C05464=1030.922,10.117,408.960,168.211,43.114,158.030
C05465=1030.915,9.868,408.976,168.209,43.115,158.030
C05466=1030.909,9.618,408.991,168.206,43.117,158.030
C05467=1030.902,9.369,409.006,168.203,43.118,158.030
C05468=1030.896,9.120,409.020,168.200,43.120,158.030
C05469=1030.890,8.870,409.035,168.199,43.121,158.030
C05470=1030.884,8.620,409.050,168.196,43.122,158.030
C05471=1030.877,8.371,409.066,168.193,43.124,158.030
C05472=1030.871,8.122,409.081,168.191,43.125,158.031
C05473=1030.864,7.872,409.096,168.189,43.126,158.031
C05474=1030.858,7.623,409.110,168.186,43.128,158.031
C05475=1030.852,7.374,409.125,168.184,43.129,158.031
C05476=1030.846,7.124,409.140,168.181,43.131,158.031
C05477=1030.839,6.874,409.155,168.179,43.132,158.031
C05478=1030.833,6.625,409.170,168.177,43.134,158.031
C05479=1030.826,6.375,409.185,168.174,43.135,158.031
C05480=1030.821,6.126,409.199,168.171,43.136,158.031
C05481=1030.814,5.876,409.214,168.169,43.138,158.031
C05482=1030.808,5.627,409.229,168.167,43.139,158.031
C05483=1030.801,5.377,409.244,168.164,43.141,158.031
C05484=1030.795,5.128,409.260,168.161,43.142,158.031
C05485=1030.789,4.879,409.275,168.159,43.143,158.031
C05486=1030.783,4.629,409.290,168.157,43.145,158.031
C05487=1030.776,4.380,409.304,168.154,43.146,158.031
C05488=1030.770,4.130,409.319,168.152,43.148,158.032
C05489=1030.764,3.881,409.334,168.150,43.149,158.032
C05490=1030.758,3.631,409.349,168.147,43.150,158.032
C05491=1030.751,3.382,409.364,168.145,43.152,158.032
C05492=1030.745,3.132,409.379,168.142,43.153,158.032
C05493=1030.739,2.883,409.393,168.139,43.154,158.032
C05494=1030.733,2.633,409.408,168.138,43.156,158.032
C05495=1030.727,2.383,409.423,168.135,43.157,158.032
C05496=1030.721,2.134,409.437,168.132,43.159,158.032
C05497=1030.715,1.885,409.452,168.129,43.160,158.032
C05498=1030.708,1.635,409.467,168.128,43.161,158.032
C05499=1030.702,1.385,409.482,168.125,43.163,158.032
C05500=1030.696,1.136,409.497,168.122,43.164,158.032
C05501=1030.690,0.887,409.512,168.120,43.165,158.032
C05502=1030.683,0.637,409.526,168.118,43.167,158.032
C05503=1030.677,0.388,409.541,168.115,43.168,158.032
C05504=1030.671,0.138,409.556,168.113,43.169,158.033
C05505=1030.665,-0.111,409.571,168.110,43.171,158.033
C05506=1030.659,-0.361,409.585,168.107,43.172,158.033
C05507=1030.653,-0.611,409.600,168.106,43.173,158.033
C05508=1030.646,-0.860,409.615,168.103,43.175,158.033
C05509=1030.641,-1.109,409.629,168.100,43.176,158.033
C05510=1030.634,-1.359,409.644,168.097,43.177,158.033
C05511=1030.628,-1.608,409.659,168.096,43.179,158.033
C05512=1030.622,-1.857,409.674,168.093,43.180,158.033
C05513=1030.616,-2.108,409.688,168.090,43.181,158.033
C05514=1030.609,-2.357,409.702,168.088,43.183,158.033
C05515=1030.603,-2.606,409.717,168.085,43.184,158.033
C05516=1030.597,-2.856,409.732,168.083,43.185,158.033
C05517=1030.591,-3.105,409.746,168.081,43.187,158.033
C05518=1030.585,-3.355,409.761,168.078,43.188,158.033
C05519=1030.578,-3.605,409.776,168.075,43.189,158.033
C05520=1030.572,-3.887,409.792,168.073,43.191,158.033
C05521=1030.565,-4.170,409.809,168.070,43.193,158.034
C05522=1030.558,-4.454,409.825,168.067,43.194,158.034
C05523=1030.550,-4.736,409.840,168.064,43.196,158.034
C05524=1030.544,-4.986,409.855,168.062,43.197,158.034
C05525=1030.538,-5.235,409.870,168.059,43.199,158.034
C05526=1030.531,-5.485,409.884,168.056,43.200,158.034
C05527=1030.525,-5.734,409.899,168.054,43.202,158.034
C05528=1030.518,-5.984,409.912,168.052,43.204,158.034
C05529=1030.512,-6.233,409.927,168.049,43.205,158.034
C05530=1030.506,-6.483,409.942,168.046,43.207,158.034
C05531=1030.500,-6.732,409.955,168.043,43.208,158.034
C05532=1030.493,-6.982,409.970,168.042,43.210,158.034
C05533=1030.487,-7.232,409.984,168.039,43.211,158.034
C05534=1030.481,-7.481,409.998,168.036,43.213,158.035
C05535=1030.475,-7.731,410.012,168.034,43.214,158.035
C05536=1030.468,-7.980,410.026,168.032,43.215,158.035
C05537=1030.462,-8.229,410.041,168.029,43.217,158.035
C05538=1030.456,-8.479,410.055,168.026,43.218,158.035
C05539=1030.449,-8.728,410.069,168.024,43.220,158.035
C05540=1030.443,-8.978,410.084,168.021,43.221,158.035
C05541=1030.437,-9.227,410.098,168.019,43.223,158.035
C05542=1030.431,-9.477,410.112,168.016,43.224,158.035
C05543=1030.424,-9.726,410.126,168.014,43.226,158.035
C05544=1030.418,-9.976,410.140,168.011,43.227,158.035
C05545=1030.412,-10.225,410.155,168.009,43.229,158.035
C05546=1030.405,-10.475,410.168,168.006,43.230,158.035
C05547=1030.400,-10.724,410.183,168.004,43.232,158.035
C05548=1030.393,-10.974,410.197,168.001,43.233,158.035
C05549=1030.387,-11.224,410.210,167.998,43.235,158.036
C05550=1030.381,-11.473,410.225,167.996,43.236,158.036
C05551=1030.375,-11.723,410.239,167.993,43.237,158.036
C05552=1030.368,-11.972,410.254,167.991,43.239,158.036
C05553=1030.362,-12.222,410.267,167.988,43.240,158.036
C05554=1030.356,-12.471,410.282,167.985,43.242,158.036
C05555=1030.349,-12.720,410.295,167.983,43.243,158.036
C05556=1030.343,-12.971,410.309,167.981,43.245,158.036
C05557=1030.338,-13.220,410.324,167.978,43.246,158.036
C05558=1030.331,-13.470,410.338,167.975,43.248,158.036
C05559=1030.325,-13.719,410.352,167.973,43.249,158.036
C05560=1030.318,-13.969,410.366,167.971,43.250,158.036
C05561=1030.313,-14.218,410.380,167.968,43.252,158.036
C05562=1030.306,-14.467,410.394,167.965,43.253,158.036
C05563=1030.300,-14.717,410.408,167.963,43.255,158.036
C05564=1030.295,-14.967,410.422,167.961,43.256,158.036
C05565=1030.288,-15.216,410.436,167.958,43.258,158.037
C05566=1030.282,-15.466,410.450,167.955,43.259,158.037
C05567=1030.275,-15.716,410.464,167.952,43.260,158.037
C05568=1030.269,-15.965,410.477,167.950,43.262,158.037
C05569=1030.263,-16.215,410.491,167.947,43.264,158.037
C05570=1030.256,-16.464,410.505,167.945,43.265,158.037
C05571=1030.250,-16.713,410.518,167.943,43.266,158.037
C05572=1030.244,-16.963,410.533,167.940,43.268,158.037
C05573=1030.238,-17.213,410.546,167.937,43.269,158.037
C05574=1030.231,-17.463,410.559,167.934,43.271,158.037
C05575=1030.225,-17.711,410.574,167.932,43.273,158.037
C05576=1030.219,-17.961,410.588,167.930,43.274,158.037
C05577=1030.212,-18.211,410.601,167.927,43.275,158.037
C05578=1030.207,-18.460,410.615,167.924,43.277,158.038
C05579=1030.200,-18.710,410.628,167.922,43.278,158.038
C05580=1030.194,-18.960,410.642,167.919,43.280,158.038
C05581=1030.187,-19.209,410.657,167.916,43.281,158.038
C05582=1030.181,-19.458,410.670,167.913,43.283,158.038
C05583=1030.175,-19.708,410.683,167.912,43.285,158.038
C05584=1030.168,-19.989,410.698,167.908,43.286,158.038
C05585=1030.161,-20.271,410.714,167.905,43.288,158.038
C05586=1030.153,-20.552,410.729,167.903,43.290,158.038
C05587=1030.147,-20.834,410.744,167.900,43.291,158.038
C05588=1030.141,-21.083,410.758,167.897,43.293,158.038
C05589=1030.134,-21.333,410.772,167.895,43.295,158.038
C05590=1030.128,-21.583,410.785,167.892,43.296,158.038
C05591=1030.122,-21.832,410.799,167.889,43.298,158.038
C05592=1030.115,-22.082,410.813,167.886,43.299,158.038
C05593=1030.109,-22.331,410.827,167.885,43.301,158.039
C05594=1030.103,-22.580,410.840,167.882,43.302,158.039
C05595=1030.098,-22.830,410.854,167.879,43.304,158.039
C05596=1030.091,-23.080,410.867,167.876,43.305,158.039
C05597=1030.085,-23.329,410.881,167.874,43.307,158.039
C05598=1030.078,-23.578,410.894,167.871,43.308,158.039
C05599=1030.072,-23.828,410.908,167.868,43.310,158.039
C05600=1030.066,-24.078,410.922,167.866,43.311,158.039
C05601=1030.060,-24.327,410.935,167.864,43.313,158.039
C05602=1030.055,-24.577,410.948,167.861,43.314,158.039
C05603=1030.048,-24.827,410.962,167.858,43.316,158.039
C05604=1030.042,-25.076,410.975,167.855,43.317,158.039
C05605=1030.035,-25.326,410.988,167.853,43.319,158.039
C05606=1030.030,-25.575,411.002,167.850,43.320,158.039
C05607=1030.023,-25.825,411.016,167.848,43.322,158.040
C05608=1030.017,-26.074,411.029,167.845,43.323,158.040
C05609=1030.011,-26.324,411.042,167.843,43.325,158.040
C05610=1030.005,-26.573,411.056,167.840,43.326,158.040
C05611=1029.998,-26.823,411.070,167.837,43.328,158.040
C05612=1029.992,-27.072,411.083,167.834,43.329,158.040
C05613=1029.986,-27.322,411.095,167.832,43.331,158.040
C05614=1029.980,-27.572,411.109,167.829,43.332,158.040
C05615=1029.973,-27.822,411.122,167.826,43.334,158.040
C05616=1029.967,-28.071,411.136,167.825,43.336,158.040
C05617=1029.961,-28.320,411.149,167.822,43.337,158.040
C05618=1029.955,-28.570,411.161,167.819,43.339,158.040
C05619=1029.948,-28.820,411.175,167.816,43.341,158.040
C05620=1029.942,-29.069,411.188,167.814,43.342,158.040
C05621=1029.936,-29.318,411.202,167.811,43.344,158.041
C05622=1029.930,-29.568,411.214,167.808,43.345,158.041
C05623=1029.924,-29.818,411.227,167.805,43.347,158.041
C05624=1029.917,-30.068,411.241,167.803,43.349,158.041
C05625=1029.910,-30.317,411.254,167.800,43.350,158.041
C05626=1029.905,-30.567,411.267,167.797,43.352,158.041
C05627=1029.898,-30.816,411.280,167.795,43.354,158.041
C05628=1029.892,-31.065,411.293,167.792,43.355,158.041
C05629=1029.886,-31.315,411.306,167.789,43.357,158.041
C05630=1029.879,-31.565,411.320,167.787,43.358,158.041
C05631=1029.873,-31.814,411.333,167.785,43.359,158.041
C05632=1029.867,-32.064,411.346,167.782,43.361,158.041
C05633=1029.861,-32.314,411.359,167.779,43.363,158.041
C05634=1029.855,-32.563,411.372,167.777,43.364,158.042
C05635=1029.849,-32.813,411.385,167.774,43.366,158.042
C05636=1029.842,-33.063,411.398,167.771,43.367,158.042
C05637=1029.836,-33.313,411.411,167.768,43.369,158.042
C05638=1029.830,-33.562,411.424,167.766,43.370,158.042
C05639=1029.824,-33.811,411.437,167.763,43.372,158.042
C05640=1029.818,-34.061,411.450,167.760,43.374,158.042
C05641=1029.812,-34.310,411.463,167.757,43.375,158.042
C05642=1029.806,-34.560,411.476,167.755,43.377,158.042
C05643=1029.800,-34.809,411.489,167.752,43.378,158.042
C05644=1029.794,-35.059,411.502,167.749,43.380,158.042
C05645=1029.787,-35.308,411.515,167.747,43.382,158.042
C05646=1029.781,-35.558,411.528,167.745,43.383,158.042
C05647=1029.775,-35.808,411.541,167.742,43.385,158.042
C05648=1029.768,-36.088,411.556,167.738,43.386,158.042
C05649=1029.761,-36.369,411.570,167.736,43.388,158.043
C05650=1029.754,-36.650,411.584,167.733,43.390,158.043
C05651=1029.747,-36.930,411.599,167.729,43.392,158.043
C05652=1029.741,-37.180,411.611,167.727,43.393,158.043
C05653=1029.735,-37.429,411.624,167.724,43.395,158.043
C05654=1029.729,-37.679,411.637,167.722,43.397,158.043
C05655=1029.723,-37.928,411.650,167.719,43.398,158.043
C05656=1029.717,-38.178,411.663,167.717,43.400,158.043
C05657=1029.711,-38.427,411.676,167.714,43.401,158.043
C05658=1029.705,-38.677,411.689,167.711,43.403,158.043
C05659=1029.699,-38.927,411.702,167.708,43.404,158.043
C05660=1029.693,-39.176,411.715,167.706,43.406,158.043
C05661=1029.686,-39.426,411.726,167.703,43.408,158.043
C05662=1029.680,-39.675,411.740,167.700,43.410,158.044
C05663=1029.674,-39.925,411.752,167.698,43.411,158.044
C05664=1029.668,-40.175,411.765,167.695,43.413,158.044
C05665=1029.661,-40.424,411.778,167.692,43.415,158.044
C05666=1029.655,-40.674,411.790,167.689,43.416,158.044
C05667=1029.649,-40.924,411.803,167.687,43.418,158.044
C05668=1029.642,-41.173,411.815,167.684,43.420,158.044
C05669=1029.636,-41.423,411.828,167.682,43.422,158.044
C05670=1029.630,-41.672,411.840,167.679,43.423,158.044
C05671=1029.624,-41.922,411.852,167.676,43.425,158.044
C05672=1029.618,-42.171,411.866,167.673,43.427,158.044
C05673=1029.612,-42.421,411.878,167.671,43.428,158.044
C05674=1029.606,-42.671,411.891,167.668,43.430,158.045
C05675=1029.599,-42.921,411.903,167.665,43.432,158.045
C05676=1029.593,-43.170,411.916,167.663,43.433,158.045
C05677=1029.587,-43.420,411.929,167.660,43.435,158.045
C05678=1029.580,-43.669,411.940,167.657,43.436,158.045
C05679=1029.574,-43.919,411.953,167.655,43.438,158.045
C05680=1029.569,-44.169,411.966,167.652,43.440,158.045
C05681=1029.562,-44.418,411.978,167.649,43.441,158.045
C05682=1029.556,-44.668,411.991,167.646,43.443,158.045
C05683=1029.550,-44.918,412.003,167.644,43.444,158.045
C05684=1029.543,-45.167,412.015,167.641,43.446,158.045
C05685=1029.538,-45.417,412.028,167.638,43.448,158.045
C05686=1029.532,-45.666,412.040,167.635,43.449,158.045
C05687=1029.525,-45.915,412.053,167.633,43.451,158.046
C05688=1029.519,-46.165,412.065,167.630,43.453,158.046
C05689=1029.513,-46.415,412.078,167.626,43.455,158.046
C05690=1029.507,-46.665,412.090,167.624,43.456,158.046
C05691=1029.501,-46.915,412.102,167.621,43.458,158.046
C05692=1029.495,-47.165,412.115,167.618,43.460,158.046
C05693=1029.489,-47.413,412.127,167.615,43.461,158.046
C05694=1029.483,-47.663,412.139,167.613,43.463,158.046
C05695=1029.477,-47.913,412.152,167.610,43.465,158.046
C05696=1029.470,-48.163,412.164,167.607,43.466,158.046
C05697=1029.464,-48.413,412.176,167.605,43.468,158.046
C05698=1029.458,-48.662,412.189,167.602,43.470,158.046
C05699=1029.452,-48.911,412.201,167.599,43.471,158.046
C05700=1029.446,-49.161,412.214,167.597,43.473,158.046
C05701=1029.439,-49.410,412.226,167.594,43.475,158.047
C05702=1029.434,-49.660,412.238,167.591,43.476,158.047
C05703=1029.428,-49.910,412.251,167.588,43.478,158.047
C05704=1029.422,-50.159,412.262,167.586,43.480,158.047
C05705=1029.416,-50.409,412.275,167.583,43.481,158.047
C05706=1029.410,-50.659,412.287,167.580,43.483,158.047
C05707=1029.403,-50.909,412.299,167.578,43.485,158.047
C05708=1029.397,-51.158,412.311,167.575,43.487,158.047
C05709=1029.391,-51.408,412.323,167.572,43.489,158.047
C05710=1029.384,-51.658,412.335,167.570,43.491,158.047
C05711=1029.378,-51.907,412.347,167.567,43.492,158.047
C05712=1029.372,-52.188,412.360,167.563,43.494,158.048
C05713=1029.364,-52.469,412.374,167.561,43.496,158.048
C05714=1029.357,-52.750,412.387,167.557,43.498,158.048
C05715=1029.350,-53.031,412.401,167.554,43.500,158.048
C05716=1029.343,-53.281,412.412,167.551,43.502,158.048
C05717=1029.338,-53.530,412.424,167.548,43.504,158.048
C05718=1029.331,-53.780,412.436,167.546,43.506,158.048
C05719=1029.325,-54.029,412.448,167.543,43.508,158.048
C05720=1029.318,-54.280,412.459,167.540,43.510,158.048
C05721=1029.313,-54.529,412.471,167.537,43.511,158.048
C05722=1029.306,-54.778,412.483,167.535,43.513,158.049
C05723=1029.300,-55.028,412.495,167.532,43.515,158.049
C05724=1029.293,-55.278,412.507,167.528,43.517,158.049
C05725=1029.288,-55.527,412.519,167.526,43.519,158.049
C05726=1029.282,-55.777,412.531,167.523,43.521,158.049
C05727=1029.275,-56.027,412.542,167.521,43.523,158.049
C05728=1029.269,-56.277,412.554,167.518,43.524,158.049
C05729=1029.263,-56.526,412.566,167.515,43.526,158.049
C05730=1029.257,-56.775,412.578,167.512,43.527,158.049
C05731=1029.250,-57.026,412.589,167.510,43.529,158.049
C05732=1029.244,-57.274,412.601,167.506,43.531,158.049
C05733=1029.238,-57.524,412.613,167.503,43.533,158.050
C05734=1029.232,-57.774,412.625,167.501,43.535,158.050
C05735=1029.226,-58.023,412.636,167.498,43.537,158.050
C05736=1029.220,-58.274,412.648,167.496,43.539,158.050
C05737=1029.214,-58.523,412.660,167.493,43.541,158.050
C05738=1029.208,-58.772,412.672,167.490,43.542,158.050
C05739=1029.201,-59.022,412.683,167.487,43.544,158.050
C05740=1029.195,-59.272,412.695,167.484,43.546,158.050
C05741=1029.190,-59.522,412.706,167.481,43.548,158.050
C05742=1029.183,-59.771,412.718,167.478,43.550,158.050
C05743=1029.176,-60.021,412.730,167.476,43.552,158.051
C05744=1029.171,-60.270,412.741,167.473,43.554,158.051
C05745=1029.164,-60.520,412.753,167.470,43.555,158.051
C05746=1029.159,-60.770,412.765,167.468,43.557,158.051
C05747=1029.152,-61.019,412.777,167.465,43.559,158.051
C05748=1029.146,-61.270,412.788,167.461,43.561,158.051
C05749=1029.140,-61.519,412.799,167.459,43.562,158.051
C05750=1029.134,-61.769,412.811,167.456,43.564,158.051
C05751=1029.128,-62.018,412.823,167.453,43.566,158.051
C05752=1029.122,-62.268,412.834,167.451,43.567,158.051
C05753=1029.115,-62.518,412.846,167.448,43.569,158.051
C05754=1029.110,-62.767,412.857,167.445,43.571,158.051
C05755=1029.104,-63.017,412.869,167.442,43.573,158.052
C05756=1029.098,-63.267,412.880,167.439,43.575,158.052
C05757=1029.091,-63.516,412.892,167.436,43.577,158.052
C05758=1029.086,-63.766,412.903,167.434,43.579,158.052
C05759=1029.079,-64.015,412.915,167.431,43.580,158.052
C05760=1029.074,-64.265,412.927,167.428,43.582,158.052
C05761=1029.068,-64.515,412.938,167.426,43.584,158.052
C05762=1029.061,-64.764,412.949,167.423,43.586,158.052
C05763=1029.055,-65.014,412.961,167.419,43.588,158.052
C05764=1029.049,-65.263,412.972,167.417,43.590,158.052
C05765=1029.043,-65.514,412.984,167.414,43.591,158.052
C05766=1029.038,-65.763,412.995,167.411,43.593,158.052
C05767=1029.031,-66.013,413.007,167.409,43.595,158.053
C05768=1029.025,-66.262,413.018,167.406,43.597,158.053
C05769=1029.019,-66.512,413.029,167.403,43.599,158.053
C05770=1029.014,-66.761,413.041,167.400,43.601,158.053
C05771=1029.007,-67.012,413.052,167.397,43.602,158.053
C05772=1029.002,-67.261,413.063,167.394,43.604,158.053
C05773=1028.995,-67.511,413.075,167.391,43.606,158.053
C05774=1028.989,-67.760,413.086,167.389,43.607,158.053
C05775=1028.983,-68.010,413.097,167.386,43.609,158.053
C05776=1028.976,-68.292,413.111,167.383,43.611,158.053
C05777=1028.970,-68.574,413.124,167.380,43.613,158.053
C05778=1028.964,-68.856,413.136,167.376,43.615,158.054
C05779=1028.956,-69.139,413.149,167.374,43.617,158.054
C05780=1028.951,-69.389,413.160,167.370,43.619,158.054
C05781=1028.945,-69.639,413.172,167.367,43.621,158.054
C05782=1028.939,-69.888,413.183,167.364,43.622,158.054
C05783=1028.932,-70.138,413.194,167.362,43.624,158.054
C05784=1028.927,-70.387,413.205,167.359,43.626,158.054
C05785=1028.921,-70.637,413.216,167.357,43.628,158.054
C05786=1028.915,-70.887,413.229,167.354,43.630,158.054
C05787=1028.909,-71.136,413.240,167.350,43.631,158.054
C05788=1028.903,-71.386,413.251,167.347,43.633,158.054
C05789=1028.897,-71.636,413.262,167.345,43.635,158.054
C05790=1028.891,-71.885,413.273,167.342,43.637,158.055
C05791=1028.885,-72.136,413.284,167.339,43.639,158.055
C05792=1028.879,-72.384,413.295,167.337,43.640,158.055
C05793=1028.874,-72.634,413.307,167.334,43.642,158.055
C05794=1028.868,-72.884,413.318,167.330,43.644,158.055
C05795=1028.862,-73.134,413.329,167.328,43.646,158.055
C05796=1028.856,-73.383,413.340,167.325,43.648,158.055
C05797=1028.850,-73.633,413.351,167.322,43.649,158.055
C05798=1028.844,-73.883,413.362,167.320,43.651,158.055
C05799=1028.838,-74.132,413.374,167.317,43.653,158.055
C05800=1028.832,-74.381,413.384,167.314,43.655,158.055
C05801=1028.826,-74.632,413.396,167.311,43.657,158.055
C05802=1028.820,-74.881,413.407,167.308,43.659,158.055
C05803=1028.815,-75.131,413.417,167.305,43.661,158.056
C05804=1028.808,-75.381,413.428,167.303,43.663,158.056
C05805=1028.803,-75.631,413.439,167.300,43.664,158.056
C05806=1028.796,-75.880,413.449,167.296,43.667,158.056
C05807=1028.790,-76.130,413.460,167.294,43.668,158.056
C05808=1028.784,-76.380,413.471,167.291,43.670,158.056
C05809=1028.778,-76.629,413.482,167.288,43.672,158.056
C05810=1028.772,-76.879,413.493,167.285,43.674,158.056
C05811=1028.766,-77.129,413.504,167.282,43.676,158.056
C05812=1028.761,-77.378,413.515,167.280,43.678,158.056
C05813=1028.754,-77.628,413.525,167.277,43.680,158.057
C05814=1028.748,-77.878,413.537,167.274,43.682,158.057
C05815=1028.742,-78.127,413.548,167.271,43.684,158.057
C05816=1028.736,-78.377,413.558,167.268,43.686,158.057
C05817=1028.731,-78.627,413.569,167.265,43.688,158.057
C05818=1028.725,-78.877,413.580,167.263,43.690,158.057
C05819=1028.719,-79.127,413.591,167.260,43.692,158.057
C05820=1028.712,-79.376,413.601,167.256,43.693,158.057
C05821=1028.707,-79.625,413.612,167.253,43.695,158.057
C05822=1028.701,-79.876,413.622,167.251,43.697,158.057
C05823=1028.695,-80.126,413.633,167.248,43.699,158.057
C05824=1028.688,-80.375,413.644,167.245,43.701,158.058
C05825=1028.683,-80.624,413.654,167.242,43.703,158.058
C05826=1028.677,-80.874,413.665,167.239,43.705,158.058
C05827=1028.670,-81.124,413.675,167.237,43.707,158.058
C05828=1028.664,-81.374,413.686,167.233,43.709,158.058
C05829=1028.658,-81.623,413.696,167.231,43.711,158.058
C05830=1028.652,-81.873,413.707,167.228,43.713,158.058
C05831=1028.646,-82.123,413.718,167.224,43.716,158.058
C05832=1028.640,-82.372,413.728,167.222,43.718,158.059
C05833=1028.634,-82.622,413.738,167.219,43.720,158.059
C05834=1028.628,-82.872,413.749,167.217,43.721,158.059
C05835=1028.622,-83.122,413.759,167.213,43.724,158.059
C05836=1028.616,-83.371,413.769,167.210,43.725,158.059
C05837=1028.609,-83.621,413.780,167.208,43.727,158.059
C05838=1028.604,-83.871,413.790,167.204,43.730,158.059
C05839=1028.598,-84.120,413.801,167.202,43.732,158.059
C05840=1028.590,-84.429,413.814,167.198,43.734,158.059
C05841=1028.582,-84.738,413.827,167.194,43.737,158.060
C05842=1028.576,-85.046,413.839,167.191,43.740,158.060
C05843=1028.568,-85.355,413.852,167.187,43.742,158.060
C05844=1028.562,-85.604,413.862,167.185,43.744,158.060
C05845=1028.556,-85.855,413.873,167.181,43.746,158.060
C05846=1028.550,-86.104,413.883,167.179,43.748,158.060
C05847=1028.544,-86.354,413.893,167.176,43.750,158.060
C05848=1028.538,-86.603,413.904,167.173,43.752,158.060
C05849=1028.532,-86.854,413.914,167.170,43.754,158.060
C05850=1028.526,-87.103,413.924,167.167,43.756,158.061
C05851=1028.520,-87.353,413.934,167.164,43.758,158.061
C05852=1028.514,-87.602,413.945,167.161,43.760,158.061
C05853=1028.508,-87.852,413.955,167.158,43.762,158.061
C05854=1028.503,-88.102,413.966,167.156,43.765,158.061
C05855=1028.497,-88.351,413.975,167.153,43.767,158.061
C05856=1028.491,-88.601,413.986,167.149,43.769,158.061
C05857=1028.485,-88.851,413.996,167.147,43.771,158.061
C05858=1028.479,-89.101,414.006,167.144,43.772,158.061
C05859=1028.473,-89.350,414.016,167.140,43.775,158.062
C05860=1028.467,-89.600,414.026,167.138,43.776,158.062
C05861=1028.461,-89.849,414.036,167.135,43.778,158.062
C05862=1028.455,-90.099,414.047,167.133,43.780,158.062
C05863=1028.449,-90.349,414.057,167.129,43.783,158.062
C05864=1028.443,-90.599,414.067,167.126,43.785,158.062
C05865=1028.437,-90.849,414.077,167.124,43.787,158.062
C05866=1028.432,-91.098,414.088,167.120,43.789,158.062
C05867=1028.425,-91.348,414.097,167.118,43.791,158.062
C05868=1028.420,-91.598,414.107,167.115,43.793,158.063
C05869=1028.413,-91.847,414.118,167.112,43.795,158.063
C05870=1028.408,-92.097,414.128,167.109,43.797,158.063
C05871=1028.402,-92.347,414.137,167.106,43.799,158.063
C05872=1028.396,-92.596,414.148,167.104,43.801,158.063
C05873=1028.391,-92.847,414.158,167.100,43.803,158.063
C05874=1028.384,-93.096,414.168,167.097,43.805,158.063
C05875=1028.379,-93.346,414.179,167.095,43.807,158.063
C05876=1028.373,-93.596,414.188,167.092,43.809,158.063
C05877=1028.367,-93.846,414.198,167.088,43.811,158.063
C05878=1028.361,-94.096,414.208,167.086,43.813,158.064
C05879=1028.355,-94.345,414.219,167.083,43.815,158.064
C05880=1028.349,-94.595,414.228,167.080,43.817,158.064
C05881=1028.344,-94.844,414.238,167.077,43.819,158.064
C05882=1028.338,-95.094,414.248,167.074,43.822,158.064
C05883=1028.332,-95.344,414.259,167.072,43.823,158.064
C05884=1028.326,-95.593,414.268,167.068,43.826,158.064
C05885=1028.320,-95.843,414.278,167.065,43.827,158.064
C05886=1028.315,-96.093,414.288,167.063,43.829,158.064
C05887=1028.308,-96.343,414.298,167.060,43.831,158.065
C05888=1028.303,-96.593,414.308,167.056,43.833,158.065
C05889=1028.297,-96.842,414.318,167.054,43.835,158.065
C05890=1028.292,-97.092,414.328,167.051,43.837,158.065
C05891=1028.285,-97.342,414.337,167.047,43.839,158.065
C05892=1028.280,-97.579,414.348,167.045,43.841,158.065
C05893=1028.274,-97.817,414.356,167.042,43.844,158.065
C05894=1028.269,-98.055,414.366,167.040,43.846,158.065
C05895=1028.264,-98.292,414.375,167.037,43.848,158.065
C05896=1028.257,-98.529,414.384,167.035,43.850,158.065
C05897=1028.252,-98.767,414.394,167.031,43.852,158.066
C05898=1028.246,-99.005,414.403,167.028,43.854,158.066
C05899=1028.241,-99.242,414.411,167.026,43.856,158.066
C05900=1028.235,-99.493,414.422,167.023,43.858,158.066
C05901=1028.230,-99.742,414.431,167.019,43.860,158.066
C05902=1028.223,-99.991,414.440,167.017,43.862,158.066
C05903=1028.217,-100.241,414.450,167.014,43.865,158.066
C05904=1028.210,-100.528,414.461,167.011,43.867,158.066
C05905=1028.203,-100.814,414.472,167.007,43.870,158.067
C05906=1028.197,-101.100,414.483,167.004,43.872,158.067
C05907=1028.190,-101.387,414.494,167.000,43.875,158.067
C05908=1028.184,-101.637,414.504,166.998,43.876,158.067
C05909=1028.178,-101.887,414.514,166.995,43.879,158.067
C05910=1028.173,-102.136,414.523,166.992,43.881,158.067
C05911=1028.167,-102.386,414.533,166.989,43.883,158.067
C05912=1028.161,-102.636,414.542,166.986,43.885,158.067
C05913=1028.155,-102.886,414.551,166.983,43.888,158.068
C05914=1028.150,-103.135,414.561,166.980,43.890,158.068
C05915=1028.144,-103.385,414.570,166.978,43.892,158.068
C05916=1028.137,-103.635,414.580,166.974,43.894,158.068
C05917=1028.131,-103.885,414.590,166.971,43.896,158.068
C05918=1028.126,-104.134,414.599,166.969,43.898,158.068
C05919=1028.120,-104.384,414.609,166.965,43.900,158.068
C05920=1028.114,-104.635,414.618,166.963,43.903,158.068
C05921=1028.109,-104.884,414.627,166.959,43.905,158.068
C05922=1028.103,-105.133,414.636,166.956,43.907,158.069
C05923=1028.097,-105.383,414.646,166.954,43.909,158.069
C05924=1028.091,-105.632,414.655,166.950,43.912,158.069
C05925=1028.086,-105.883,414.665,166.948,43.914,158.069
C05926=1028.080,-106.133,414.674,166.945,43.916,158.069
C05927=1028.074,-106.382,414.683,166.942,43.918,158.069
C05928=1028.068,-106.632,414.693,166.939,43.920,158.069
C05929=1028.062,-106.882,414.702,166.936,43.922,158.069
C05930=1028.056,-107.131,414.711,166.933,43.925,158.070
C05931=1028.050,-107.381,414.721,166.930,43.927,158.070
C05932=1028.044,-107.631,414.730,166.928,43.929,158.070
C05933=1028.039,-107.881,414.739,166.924,43.932,158.070
C05934=1028.033,-108.130,414.748,166.922,43.934,158.070
C05935=1028.027,-108.380,414.758,166.918,43.936,158.070
C05936=1028.021,-108.630,414.766,166.916,43.938,158.070
C05937=1028.015,-108.880,414.776,166.913,43.940,158.070
C05938=1028.009,-109.130,414.785,166.909,43.943,158.071
C05939=1028.004,-109.379,414.794,166.907,43.945,158.071
C05940=1027.997,-109.629,414.804,166.903,43.947,158.071
C05941=1027.992,-109.879,414.812,166.901,43.950,158.071
C05942=1027.986,-110.128,414.822,166.898,43.952,158.071
C05943=1027.980,-110.379,414.830,166.895,43.954,158.071
C05944=1027.975,-110.628,414.840,166.892,43.956,158.071
C05945=1027.968,-110.878,414.849,166.889,43.958,158.072
C05946=1027.963,-111.128,414.858,166.886,43.961,158.072
C05947=1027.957,-111.377,414.867,166.883,43.963,158.072
C05948=1027.952,-111.627,414.876,166.880,43.965,158.072
C05949=1027.946,-111.877,414.885,166.877,43.968,158.072
C05950=1027.940,-112.127,414.894,166.875,43.970,158.072
C05951=1027.934,-112.376,414.903,166.871,43.972,158.072
C05952=1027.928,-112.627,414.912,166.869,43.974,158.072
C05953=1027.923,-112.876,414.921,166.866,43.976,158.073
C05954=1027.917,-113.126,414.930,166.862,43.979,158.073
C05955=1027.911,-113.375,414.939,166.860,43.981,158.073
C05956=1027.905,-113.626,414.948,166.856,43.984,158.073
C05957=1027.900,-113.875,414.957,166.854,43.986,158.073
C05958=1027.894,-114.125,414.966,166.851,43.988,158.073
C05959=1027.888,-114.374,414.976,166.848,43.990,158.073
C05960=1027.883,-114.625,414.984,166.845,43.992,158.073
C05961=1027.877,-114.874,414.992,166.842,43.995,158.074
C05962=1027.870,-115.124,415.002,166.839,43.997,158.074
C05963=1027.865,-115.374,415.010,166.837,44.000,158.074
C05964=1027.859,-115.624,415.020,166.833,44.002,158.074
C05965=1027.854,-115.873,415.028,166.830,44.004,158.074
C05966=1027.848,-116.124,415.037,166.827,44.007,158.074
C05967=1027.841,-116.372,415.046,166.824,44.008,158.074
C05968=1027.836,-116.659,415.056,166.821,44.011,158.075
C05969=1027.828,-116.945,415.066,166.817,44.014,158.075
C05970=1027.822,-117.231,415.076,166.814,44.017,158.075
C05971=1027.815,-117.517,415.086,166.810,44.020,158.075
C05972=1027.809,-117.767,415.095,166.808,44.022,158.075
C05973=1027.804,-118.017,415.104,166.805,44.024,158.075
C05974=1027.799,-118.267,415.112,166.802,44.026,158.075
C05975=1027.792,-118.516,415.121,166.799,44.029,158.076
C05976=1027.787,-118.766,415.130,166.796,44.031,158.076
C05977=1027.781,-119.016,415.138,166.793,44.034,158.076
C05978=1027.776,-119.266,415.147,166.791,44.036,158.076
C05979=1027.769,-119.515,415.156,166.787,44.038,158.076
C05980=1027.763,-119.765,415.164,166.784,44.040,158.076
C05981=1027.758,-120.015,415.173,166.781,44.043,158.076
C05982=1027.752,-120.265,415.182,166.778,44.045,158.077
C05983=1027.746,-120.515,415.190,166.775,44.048,158.077
C05984=1027.741,-120.764,415.199,166.772,44.050,158.077
C05985=1027.735,-121.014,415.208,166.770,44.053,158.077
C05986=1027.730,-121.264,415.216,166.766,44.055,158.077
C05987=1027.724,-121.513,415.224,166.764,44.057,158.077
C05988=1027.718,-121.764,415.233,166.760,44.059,158.077
C05989=1027.712,-122.013,415.241,166.758,44.062,158.078
C05990=1027.706,-122.263,415.251,166.755,44.064,158.078
C05991=1027.700,-122.513,415.259,166.752,44.067,158.078
C05992=1027.695,-122.762,415.267,166.749,44.069,158.078
C05993=1027.690,-123.012,415.276,166.746,44.072,158.078
C05994=1027.684,-123.262,415.285,166.743,44.073,158.078
C05995=1027.678,-123.512,415.293,166.740,44.076,158.078
C05996=1027.673,-123.762,415.301,166.737,44.078,158.079
C05997=1027.667,-124.012,415.310,166.735,44.081,158.079
C05998=1027.661,-124.261,415.318,166.731,44.083,158.079
C05999=1027.655,-124.511,415.326,166.728,44.086,158.079
C06000=1027.650,-124.762,415.335,166.725,44.088,158.079
C06001=1027.644,-125.011,415.343,166.722,44.090,158.079
C06002=1027.638,-125.261,415.351,166.719,44.093,158.079
C06003=1027.632,-125.511,415.360,166.716,44.095,158.080
C06004=1027.626,-125.760,415.368,166.714,44.098,158.080
C06005=1027.621,-126.010,415.377,166.710,44.101,158.080
C06006=1027.615,-126.260,415.385,166.708,44.102,158.080
C06007=1027.609,-126.510,415.393,166.704,44.105,158.080
C06008=1027.603,-126.759,415.401,166.702,44.108,158.080
C06009=1027.598,-127.009,415.410,166.698,44.110,158.080
C06010=1027.592,-127.259,415.418,166.696,44.113,158.081
C06011=1027.586,-127.509,415.427,166.693,44.115,158.081
C06012=1027.581,-127.758,415.434,166.690,44.117,158.081
C06013=1027.576,-128.007,415.443,166.687,44.119,158.081
C06014=1027.571,-128.257,415.452,166.685,44.121,158.081
C06015=1027.566,-128.507,415.461,166.682,44.123,158.081
C06016=1027.562,-128.757,415.472,166.679,44.124,158.081
C06017=1027.559,-129.006,415.482,166.676,44.124,158.081
C06018=1027.556,-129.256,415.493,166.674,44.124,158.081
C06019=1027.555,-129.506,415.505,166.671,44.124,158.080
C06020=1027.552,-129.756,415.518,166.669,44.123,158.080
C06021=1027.552,-130.006,415.531,166.667,44.121,158.080
C06022=1027.551,-130.255,415.544,166.665,44.120,158.079
C06023=1027.552,-130.505,415.558,166.663,44.117,158.079
C06024=1027.553,-130.755,415.573,166.661,44.115,158.078
C06025=1027.554,-131.005,415.588,166.659,44.111,158.077
C06026=1027.556,-131.255,415.604,166.657,44.107,158.076
C06027=1027.559,-131.505,415.621,166.655,44.103,158.075
C06028=1027.562,-131.754,415.638,166.653,44.098,158.075
C06029=1027.565,-132.005,415.655,166.652,44.093,158.074
C06030=1027.570,-132.254,415.673,166.651,44.087,158.073
C06031=1027.574,-132.504,415.693,166.649,44.081,158.071
C06032=1027.264,-132.529,415.376,166.601,44.336,158.110
C06033=1027.260,-132.280,415.357,166.603,44.342,158.111
C06034=1027.256,-132.030,415.339,166.604,44.348,158.112
C06035=1027.252,-131.781,415.321,166.605,44.353,158.113
C06036=1027.249,-131.530,415.304,166.607,44.358,158.114
C06037=1027.246,-131.280,415.288,166.608,44.362,158.115
C06038=1027.244,-131.031,415.272,166.611,44.366,158.115
C06039=1027.243,-130.781,415.256,166.613,44.369,158.116
C06040=1027.241,-130.530,415.242,166.615,44.372,158.117
C06041=1027.242,-130.281,415.227,166.617,44.374,158.117
C06042=1027.242,-130.031,415.213,166.618,44.376,158.118
C06043=1027.243,-129.781,415.200,166.621,44.377,158.118
C06044=1027.244,-129.531,415.188,166.623,44.378,158.119
C06045=1027.246,-129.281,415.176,166.626,44.379,158.119
C06046=1027.249,-129.032,415.165,166.628,44.379,158.119
C06047=1027.252,-128.782,415.154,166.630,44.379,158.119
C06048=1027.256,-128.533,415.144,166.633,44.377,158.119
C06049=1027.260,-128.283,415.135,166.636,44.376,158.119
C06050=1027.265,-128.033,415.126,166.638,44.374,158.119
C06051=1027.271,-127.784,415.117,166.642,44.372,158.119
C06052=1027.277,-127.534,415.109,166.644,44.369,158.119
C06053=1027.282,-127.285,415.100,166.648,44.366,158.119
C06054=1027.287,-127.035,415.093,166.650,44.364,158.119
C06055=1027.293,-126.785,415.085,166.654,44.362,158.119
C06056=1027.299,-126.535,415.076,166.656,44.359,158.118
C06057=1027.305,-126.285,415.068,166.660,44.357,158.118
C06058=1027.310,-126.035,415.059,166.662,44.354,158.118
C06059=1027.316,-125.786,415.051,166.665,44.352,158.118
C06060=1027.322,-125.535,415.043,166.668,44.349,158.118
C06061=1027.328,-125.286,415.035,166.671,44.347,158.118
C06062=1027.333,-125.036,415.026,166.674,44.345,158.118
C06063=1027.339,-124.787,415.018,166.677,44.342,158.117
C06064=1027.345,-124.537,415.009,166.680,44.339,158.117
C06065=1027.350,-124.287,415.001,166.683,44.337,158.117
C06066=1027.356,-124.037,414.993,166.686,44.334,158.117
C06067=1027.362,-123.787,414.984,166.689,44.332,158.117
C06068=1027.367,-123.537,414.976,166.692,44.329,158.117
C06069=1027.373,-123.288,414.967,166.695,44.327,158.117
C06070=1027.379,-123.037,414.959,166.698,44.325,158.117
C06071=1027.384,-122.788,414.951,166.701,44.322,158.116
C06072=1027.390,-122.538,414.942,166.703,44.320,158.116
C06073=1027.396,-122.289,414.934,166.707,44.317,158.116
C06074=1027.402,-122.039,414.925,166.709,44.315,158.116
C06075=1027.407,-121.789,414.916,166.713,44.312,158.116
C06076=1027.412,-121.539,414.908,166.715,44.310,158.116
C06077=1027.419,-121.289,414.899,166.719,44.308,158.116
C06078=1027.424,-121.040,414.891,166.721,44.305,158.115
C06079=1027.430,-120.790,414.882,166.725,44.303,158.115
C06080=1027.435,-120.539,414.874,166.727,44.300,158.115
C06081=1027.442,-120.291,414.865,166.730,44.298,158.115
C06082=1027.448,-120.040,414.856,166.733,44.295,158.115
C06083=1027.453,-119.791,414.848,166.736,44.293,158.115
C06084=1027.458,-119.541,414.839,166.740,44.291,158.115
C06085=1027.465,-119.291,414.831,166.742,44.288,158.114
C06086=1027.470,-119.042,414.822,166.746,44.286,158.114
C06087=1027.476,-118.792,414.813,166.748,44.283,158.114
C06088=1027.481,-118.541,414.804,166.751,44.281,158.114
C06089=1027.487,-118.292,414.796,166.754,44.278,158.114
C06090=1027.494,-118.042,414.787,166.757,44.276,158.114
C06091=1027.499,-117.793,414.778,166.760,44.274,158.114
C06092=1027.505,-117.542,414.770,166.763,44.272,158.113
C06093=1027.512,-117.257,414.760,166.766,44.269,158.113
C06094=1027.517,-116.970,414.750,166.770,44.266,158.113
C06095=1027.524,-116.684,414.740,166.773,44.263,158.113
C06096=1027.531,-116.399,414.730,166.776,44.260,158.113
C06097=1027.537,-116.148,414.721,166.779,44.258,158.113
C06098=1027.542,-115.899,414.712,166.782,44.256,158.112
C06099=1027.548,-115.649,414.703,166.785,44.254,158.112
C06100=1027.554,-115.399,414.695,166.789,44.251,158.112
C06101=1027.560,-115.149,414.685,166.791,44.249,158.112
C06102=1027.566,-114.900,414.677,166.795,44.246,158.112
C06103=1027.572,-114.650,414.668,166.797,44.244,158.112
C06104=1027.577,-114.401,414.659,166.800,44.241,158.112
C06105=1027.583,-114.150,414.650,166.803,44.239,158.112
C06106=1027.589,-113.901,414.641,166.806,44.237,158.111
C06107=1027.595,-113.651,414.632,166.809,44.234,158.111
C06108=1027.600,-113.401,414.623,166.812,44.232,158.111
C06109=1027.606,-113.151,414.614,166.814,44.230,158.111
C06110=1027.611,-112.901,414.606,166.818,44.227,158.111
C06111=1027.617,-112.652,414.596,166.820,44.225,158.111
C06112=1027.623,-112.402,414.588,166.824,44.223,158.111
C06113=1027.629,-112.152,414.578,166.826,44.220,158.110
C06114=1027.634,-111.902,414.570,166.830,44.218,158.110
C06115=1027.640,-111.653,414.560,166.832,44.216,158.110
C06116=1027.646,-111.403,414.551,166.835,44.214,158.110
C06117=1027.652,-111.153,414.542,166.839,44.211,158.110
C06118=1027.657,-110.904,414.533,166.841,44.209,158.110
C06119=1027.663,-110.653,414.524,166.845,44.206,158.110
C06120=1027.669,-110.404,414.514,166.847,44.204,158.110
C06121=1027.675,-110.154,414.506,166.850,44.202,158.109
C06122=1027.681,-109.904,414.496,166.853,44.199,158.109
C06123=1027.686,-109.654,414.488,166.856,44.197,158.109
C06124=1027.693,-109.405,414.479,166.859,44.195,158.109
C06125=1027.699,-109.155,414.469,166.862,44.193,158.109
C06126=1027.704,-108.905,414.461,166.864,44.190,158.109
C06127=1027.711,-108.656,414.451,166.868,44.188,158.109
C06128=1027.716,-108.406,414.443,166.870,44.185,158.108
C06129=1027.722,-108.156,414.433,166.874,44.183,158.108
C06130=1027.728,-107.906,414.424,166.877,44.181,158.108
C06131=1027.733,-107.657,414.415,166.880,44.178,158.108
C06132=1027.739,-107.407,414.405,166.883,44.176,158.108
C06133=1027.745,-107.157,414.395,166.885,44.174,158.108
C06134=1027.750,-106.907,414.387,166.889,44.172,158.108
C06135=1027.756,-106.657,414.377,166.891,44.170,158.108
C06136=1027.762,-106.408,414.368,166.894,44.167,158.107
C06137=1027.768,-106.158,414.359,166.897,44.165,158.107
C06138=1027.774,-105.908,414.350,166.900,44.163,158.107
C06139=1027.780,-105.659,414.341,166.904,44.160,158.107
C06140=1027.786,-105.409,414.331,166.906,44.158,158.107
C06141=1027.791,-105.159,414.321,166.909,44.156,158.107
C06142=1027.797,-104.910,414.312,166.912,44.153,158.107
C06143=1027.803,-104.659,414.303,166.915,44.152,158.107
C06144=1027.809,-104.410,414.293,166.919,44.149,158.107
C06145=1027.815,-104.160,414.284,166.921,44.147,158.106
C06146=1027.821,-103.911,414.274,166.924,44.145,158.106
C06147=1027.826,-103.661,414.264,166.927,44.143,158.106
C06148=1027.832,-103.410,414.255,166.930,44.140,158.106
C06149=1027.837,-103.161,414.246,166.932,44.138,158.106
C06150=1027.844,-102.911,414.237,166.936,44.136,158.106
C06151=1027.850,-102.661,414.227,166.938,44.133,158.106
C06152=1027.855,-102.411,414.217,166.942,44.131,158.106
C06153=1027.861,-102.162,414.208,166.945,44.129,158.105
C06154=1027.867,-101.912,414.198,166.947,44.127,158.105
C06155=1027.873,-101.663,414.189,166.951,44.125,158.105
C06156=1027.879,-101.413,414.179,166.953,44.123,158.105
C06157=1027.885,-101.127,414.168,166.957,44.120,158.105
C06158=1027.892,-100.840,414.158,166.960,44.117,158.105
C06159=1027.899,-100.554,414.147,166.964,44.115,158.105
C06160=1027.906,-100.267,414.136,166.967,44.112,158.105
C06161=1027.911,-100.017,414.126,166.970,44.110,158.104
C06162=1027.917,-99.767,414.116,166.972,44.108,158.104
C06163=1027.923,-99.517,414.107,166.976,44.105,158.104
C06164=1027.929,-99.268,414.097,166.978,44.103,158.104
C06165=1027.934,-99.018,414.087,166.981,44.101,158.104
C06166=1027.940,-98.768,414.078,166.985,44.099,158.104
C06167=1027.947,-98.519,414.068,166.987,44.097,158.104
C06168=1027.953,-98.269,414.059,166.990,44.094,158.103
C06169=1027.959,-98.019,414.049,166.993,44.092,158.103
C06170=1027.964,-97.769,414.039,166.996,44.090,158.103
C06171=1027.970,-97.520,414.030,167.000,44.088,158.103
C06172=1027.975,-97.270,414.019,167.002,44.085,158.103
C06173=1027.982,-97.021,414.009,167.005,44.083,158.103
C06174=1027.987,-96.770,413.999,167.008,44.081,158.103
C06175=1027.994,-96.521,413.989,167.011,44.079,158.103
C06176=1028.000,-96.271,413.980,167.013,44.077,158.103
C06177=1028.005,-96.021,413.970,167.016,44.076,158.103
C06178=1028.011,-95.772,413.960,167.020,44.073,158.103
C06179=1028.016,-95.522,413.950,167.022,44.071,158.102
C06180=1028.023,-95.272,413.940,167.025,44.069,158.102
C06181=1028.028,-95.022,413.930,167.028,44.067,158.102
C06182=1028.034,-94.772,413.920,167.031,44.065,158.102
C06183=1028.040,-94.522,413.910,167.034,44.063,158.102
C06184=1028.046,-94.273,413.900,167.037,44.061,158.102
C06185=1028.051,-94.024,413.890,167.040,44.058,158.102
C06186=1028.057,-93.774,413.881,167.042,44.056,158.102
C06187=1028.063,-93.524,413.870,167.046,44.054,158.102
C06188=1028.069,-93.275,413.860,167.049,44.052,158.101
C06189=1028.074,-93.025,413.850,167.051,44.050,158.101
C06190=1028.081,-92.775,413.840,167.054,44.048,158.101
C06191=1028.086,-92.525,413.829,167.058,44.046,158.101
C06192=1028.093,-92.275,413.820,167.060,44.044,158.101
C06193=1028.098,-92.025,413.810,167.063,44.042,158.101
C06194=1028.104,-91.776,413.799,167.066,44.040,158.101
C06195=1028.110,-91.526,413.789,167.069,44.038,158.101
C06196=1028.116,-91.276,413.780,167.072,44.036,158.101
C06197=1028.122,-91.027,413.769,167.075,44.034,158.101
C06198=1028.128,-90.777,413.759,167.078,44.031,158.100
C06199=1028.133,-90.527,413.749,167.080,44.029,158.100
C06200=1028.139,-90.277,413.738,167.084,44.027,158.100
C06201=1028.145,-90.028,413.729,167.086,44.025,158.100
C06202=1028.151,-89.777,413.719,167.089,44.023,158.100
C06203=1028.157,-89.528,413.708,167.093,44.021,158.100
C06204=1028.163,-89.278,413.698,167.095,44.018,158.100
C06205=1028.169,-89.029,413.688,167.098,44.016,158.100
C06206=1028.175,-88.779,413.678,167.100,44.015,158.099
C06207=1028.181,-88.529,413.668,167.104,44.012,158.099
C06208=1028.186,-88.280,413.657,167.107,44.010,158.099
C06209=1028.193,-88.030,413.648,167.109,44.009,158.099
C06210=1028.198,-87.780,413.637,167.113,44.006,158.099
C06211=1028.205,-87.531,413.627,167.115,44.004,158.099
C06212=1028.210,-87.281,413.616,167.118,44.002,158.099
C06213=1028.216,-87.031,413.607,167.122,44.000,158.099
C06214=1028.222,-86.782,413.596,167.124,43.998,158.099
C06215=1028.228,-86.532,413.586,167.127,43.995,158.098
C06216=1028.234,-86.282,413.575,167.130,43.993,158.098
C06217=1028.240,-86.032,413.565,167.133,43.991,158.098
C06218=1028.246,-85.783,413.555,167.136,43.989,158.098
C06219=1028.251,-85.533,413.545,167.138,43.987,158.098
C06220=1028.258,-85.284,413.535,167.142,43.985,158.098
C06221=1028.265,-84.999,413.523,167.145,43.982,158.098
C06222=1028.271,-84.715,413.511,167.148,43.981,158.098
C06223=1028.279,-84.430,413.499,167.151,43.978,158.098
C06224=1028.286,-84.146,413.487,167.155,43.976,158.098
C06225=1028.291,-83.896,413.476,167.157,43.973,158.097
C06226=1028.298,-83.647,413.466,167.160,43.971,158.097
C06227=1028.303,-83.397,413.456,167.164,43.969,158.097
C06228=1028.310,-83.148,413.446,167.166,43.967,158.097
C06229=1028.317,-82.823,413.432,167.170,43.964,158.097
C06230=1028.325,-82.497,413.419,167.174,43.961,158.097
C06231=1028.333,-82.172,413.405,167.178,43.959,158.097
C06232=1028.341,-81.848,413.391,167.181,43.956,158.096
C06233=1028.346,-81.598,413.381,167.185,43.954,158.096
C06234=1028.353,-81.348,413.370,167.187,43.952,158.096
C06235=1028.359,-81.098,413.359,167.190,43.950,158.096
C06236=1028.365,-80.848,413.350,167.194,43.948,158.096
C06237=1028.371,-80.599,413.339,167.196,43.945,158.096
C06238=1028.377,-80.349,413.328,167.199,43.943,158.096
C06239=1028.384,-80.099,413.318,167.202,43.941,158.096
C06240=1028.389,-79.849,413.307,167.205,43.939,158.096
C06241=1028.395,-79.600,413.296,167.208,43.937,158.095
C06242=1028.401,-79.350,413.285,167.210,43.935,158.095
C06243=1028.408,-79.101,413.275,167.214,43.933,158.095
C06244=1028.413,-78.850,413.265,167.217,43.931,158.095
C06245=1028.419,-78.601,413.254,167.219,43.929,158.095
C06246=1028.425,-78.352,413.243,167.222,43.927,158.095
C06247=1028.430,-78.102,413.232,167.224,43.926,158.095
C06248=1028.437,-77.852,413.221,167.228,43.923,158.095
C06249=1028.443,-77.603,413.210,167.231,43.922,158.095
C06250=1028.449,-77.353,413.200,167.233,43.920,158.095
C06251=1028.455,-77.104,413.189,167.236,43.918,158.094
C06252=1028.461,-76.853,413.178,167.240,43.916,158.094
C06253=1028.467,-76.603,413.167,167.242,43.914,158.094
C06254=1028.472,-76.354,413.156,167.245,43.912,158.094
C06255=1028.479,-76.104,413.145,167.247,43.909,158.094
C06256=1028.485,-75.855,413.135,167.251,43.907,158.094
C06257=1028.491,-75.605,413.124,167.254,43.905,158.094
C06258=1028.497,-75.356,413.113,167.256,43.903,158.094
C06259=1028.503,-75.105,413.102,167.259,43.901,158.094
C06260=1028.509,-74.856,413.091,167.263,43.899,158.094
C06261=1028.514,-74.606,413.080,167.265,43.897,158.093
C06262=1028.521,-74.356,413.069,167.268,43.895,158.093
C06263=1028.527,-74.107,413.059,167.270,43.894,158.093
C06264=1028.532,-73.857,413.047,167.274,43.891,158.093
C06265=1028.539,-73.607,413.036,167.277,43.889,158.093
C06266=1028.544,-73.358,413.025,167.280,43.888,158.093
C06267=1028.550,-73.108,413.014,167.282,43.886,158.093
C06268=1028.556,-72.858,413.003,167.285,43.884,158.093
C06269=1028.562,-72.608,412.992,167.287,43.883,158.093
C06270=1028.568,-72.359,412.980,167.291,43.880,158.093
C06271=1028.573,-72.110,412.969,167.294,43.879,158.093
C06272=1028.580,-71.859,412.958,167.297,43.877,158.093
C06273=1028.585,-71.610,412.947,167.299,43.875,158.092
C06274=1028.591,-71.360,412.936,167.302,43.873,158.092
C06275=1028.597,-71.110,412.925,167.304,43.872,158.092
C06276=1028.603,-70.861,412.913,167.308,43.869,158.092
C06277=1028.610,-70.611,412.902,167.311,43.868,158.092
C06278=1028.615,-70.361,412.890,167.313,43.866,158.092
C06279=1028.620,-70.112,412.880,167.316,43.864,158.092
C06280=1028.627,-69.862,412.868,167.319,43.863,158.092
C06281=1028.632,-69.634,412.858,167.321,43.861,158.092
C06282=1028.638,-69.406,412.848,167.324,43.859,158.092
C06283=1028.643,-69.178,412.837,167.327,43.857,158.092
C06284=1028.649,-68.949,412.826,167.330,43.856,158.092
C06285=1028.654,-68.721,412.817,167.332,43.854,158.092
C06286=1028.660,-68.492,412.806,167.335,43.852,158.091
C06287=1028.665,-68.265,412.796,167.337,43.851,158.091
C06288=1028.670,-68.036,412.785,167.339,43.849,158.091
C06289=1028.676,-67.786,412.774,167.343,43.847,158.091
C06290=1028.682,-67.537,412.762,167.346,43.845,158.091
C06291=1028.688,-67.287,412.752,167.348,43.843,158.091
C06292=1028.695,-67.037,412.740,167.351,43.841,158.091
C06293=1028.701,-66.788,412.729,167.354,43.839,158.091
C06294=1028.706,-66.538,412.717,167.356,43.838,158.091
C06295=1028.712,-66.288,412.706,167.360,43.836,158.091
C06296=1028.718,-66.039,412.694,167.363,43.834,158.091
C06297=1028.724,-65.789,412.683,167.365,43.832,158.091
C06298=1028.730,-65.540,412.672,167.368,43.830,158.090
C06299=1028.736,-65.290,412.660,167.371,43.828,158.090
C06300=1028.742,-65.040,412.649,167.373,43.826,158.090
C06301=1028.748,-64.790,412.638,167.377,43.824,158.090
C06302=1028.754,-64.541,412.626,167.379,43.822,158.090
C06303=1028.760,-64.291,412.615,167.382,43.821,158.090
C06304=1028.766,-64.042,412.603,167.385,43.819,158.090
C06305=1028.772,-63.792,412.591,167.388,43.817,158.090
C06306=1028.778,-63.542,412.580,167.390,43.815,158.090
C06307=1028.784,-63.293,412.568,167.394,43.813,158.090
C06308=1028.791,-63.042,412.557,167.396,43.811,158.090
C06309=1028.796,-62.793,412.545,167.399,43.809,158.089
C06310=1028.802,-62.543,412.534,167.402,43.807,158.089
C06311=1028.808,-62.294,412.522,167.404,43.806,158.089
C06312=1028.815,-62.044,412.511,167.407,43.804,158.089
C06313=1028.821,-61.795,412.499,167.410,43.802,158.089
C06314=1028.826,-61.545,412.488,167.413,43.800,158.089
C06315=1028.832,-61.296,412.476,167.416,43.798,158.089
C06316=1028.839,-61.046,412.465,167.419,43.797,158.089
C06317=1028.845,-60.796,412.453,167.421,43.795,158.089
C06318=1028.851,-60.546,412.442,167.424,43.793,158.089
C06319=1028.857,-60.297,412.429,167.427,43.791,158.089
C06320=1028.863,-60.047,412.418,167.430,43.789,158.088
C06321=1028.870,-59.798,412.406,167.433,43.787,158.088
C06322=1028.876,-59.547,412.395,167.436,43.785,158.088
C06323=1028.881,-59.298,412.383,167.438,43.783,158.088
C06324=1028.888,-59.049,412.371,167.441,43.781,158.088
C06325=1028.894,-58.798,412.360,167.443,43.779,158.088
C06326=1028.900,-58.550,412.348,167.447,43.777,158.088
C06327=1028.907,-58.299,412.337,167.450,43.775,158.088
C06328=1028.912,-58.049,412.324,167.452,43.773,158.088
C06329=1028.918,-57.801,412.313,167.455,43.772,158.088
C06330=1028.925,-57.550,412.302,167.458,43.770,158.088
C06331=1028.931,-57.301,412.290,167.461,43.768,158.087
C06332=1028.936,-57.051,412.278,167.464,43.766,158.087
C06333=1028.943,-56.801,412.266,167.467,43.764,158.087
C06334=1028.950,-56.552,412.254,167.469,43.762,158.087
C06335=1028.956,-56.302,412.243,167.472,43.761,158.087
C06336=1028.961,-56.052,412.231,167.475,43.759,158.087
C06337=1028.968,-55.803,412.219,167.477,43.757,158.087
C06338=1028.974,-55.553,412.208,167.480,43.755,158.087
C06339=1028.980,-55.304,412.196,167.484,43.753,158.087
C06340=1028.986,-55.054,412.183,167.486,43.751,158.086
C06341=1028.993,-54.804,412.172,167.489,43.749,158.086
C06342=1028.999,-54.555,412.161,167.492,43.747,158.086
C06343=1029.005,-54.305,412.149,167.494,43.745,158.086
C06344=1029.011,-54.055,412.136,167.497,43.743,158.086
C06345=1029.018,-53.805,412.125,167.500,43.741,158.086
C06346=1029.024,-53.556,412.113,167.503,43.739,158.086
C06347=1029.030,-53.307,412.101,167.506,43.737,158.086
C06348=1029.036,-53.057,412.089,167.508,43.735,158.086
C06349=1029.043,-52.776,412.076,167.512,43.733,158.086
C06350=1029.050,-52.495,412.062,167.515,43.732,158.085
C06351=1029.057,-52.214,412.049,167.518,43.729,158.085
C06352=1029.064,-51.933,412.035,167.521,43.727,158.085
C06353=1029.070,-51.683,412.024,167.523,43.725,158.085
C06354=1029.077,-51.434,412.012,167.526,43.723,158.085
C06355=1029.084,-51.184,412.000,167.530,43.721,158.085
C06356=1029.089,-50.935,411.988,167.532,43.719,158.085
C06357=1029.096,-50.685,411.976,167.535,43.717,158.085
C06358=1029.102,-50.435,411.963,167.538,43.716,158.085
C06359=1029.108,-50.186,411.951,167.540,43.714,158.085
C06360=1029.114,-49.936,411.939,167.543,43.712,158.084
C06361=1029.120,-49.686,411.926,167.546,43.710,158.084
C06362=1029.126,-49.437,411.915,167.548,43.709,158.084
C06363=1029.132,-49.187,411.902,167.551,43.707,158.084
C06364=1029.139,-48.938,411.890,167.554,43.705,158.084
C06365=1029.145,-48.688,411.878,167.557,43.704,158.084
C06366=1029.151,-48.438,411.865,167.559,43.702,158.084
C06367=1029.157,-48.189,411.853,167.562,43.700,158.084
C06368=1029.162,-47.939,411.841,167.565,43.698,158.084
C06369=1029.168,-47.689,411.828,167.568,43.697,158.084
C06370=1029.175,-47.440,411.816,167.571,43.695,158.084
C06371=1029.181,-47.190,411.804,167.574,43.693,158.084
C06372=1029.187,-46.940,411.791,167.576,43.691,158.083
C06373=1029.193,-46.691,411.780,167.579,43.690,158.084
C06374=1029.199,-46.441,411.767,167.582,43.688,158.083
C06375=1029.205,-46.191,411.755,167.584,43.686,158.083
C06376=1029.211,-45.942,411.743,167.587,43.684,158.083
C06377=1029.218,-45.693,411.729,167.590,43.683,158.083
C06378=1029.223,-45.443,411.717,167.592,43.681,158.083
C06379=1029.230,-45.193,411.705,167.595,43.679,158.083
C06380=1029.236,-44.943,411.692,167.598,43.678,158.083
C06381=1029.241,-44.694,411.680,167.600,43.676,158.083
C06382=1029.248,-44.445,411.668,167.603,43.674,158.083
C06383=1029.254,-44.195,411.656,167.606,43.673,158.083
C06384=1029.260,-43.945,411.642,167.608,43.671,158.083
C06385=1029.267,-43.696,411.630,167.611,43.669,158.082
C06386=1029.273,-43.446,411.618,167.614,43.668,158.082
C06387=1029.279,-43.196,411.605,167.617,43.666,158.082
C06388=1029.285,-42.946,411.593,167.620,43.664,158.082
C06389=1029.291,-42.697,411.580,167.623,43.662,158.082
C06390=1029.297,-42.447,411.567,167.626,43.660,158.082
C06391=1029.304,-42.198,411.555,167.628,43.659,158.082
C06392=1029.310,-41.948,411.543,167.631,43.657,158.082
C06393=1029.316,-41.699,411.530,167.634,43.655,158.082
C06394=1029.323,-41.449,411.518,167.636,43.653,158.082
C06395=1029.329,-41.199,411.505,167.639,43.651,158.082
C06396=1029.335,-40.949,411.493,167.642,43.650,158.082
C06397=1029.341,-40.700,411.479,167.644,43.648,158.081
C06398=1029.347,-40.450,411.467,167.647,43.646,158.081
C06399=1029.353,-40.201,411.455,167.650,43.644,158.081
C06400=1029.360,-39.951,411.442,167.652,43.642,158.081
C06401=1029.366,-39.702,411.430,167.655,43.641,158.081
C06402=1029.372,-39.452,411.417,167.658,43.639,158.081
C06403=1029.378,-39.202,411.404,167.660,43.637,158.081
C06404=1029.385,-38.953,411.392,167.663,43.635,158.081
C06405=1029.391,-38.703,411.379,167.666,43.634,158.081
C06406=1029.397,-38.454,411.366,167.669,43.632,158.081
C06407=1029.403,-38.204,411.353,167.671,43.630,158.081
C06408=1029.409,-37.955,411.340,167.674,43.629,158.081
C06409=1029.415,-37.705,411.328,167.677,43.627,158.080
C06410=1029.421,-37.455,411.315,167.679,43.625,158.080
C06411=1029.427,-37.206,411.302,167.682,43.624,158.080
C06412=1029.433,-36.956,411.289,167.685,43.622,158.080
C06413=1029.440,-36.676,411.274,167.687,43.620,158.080
C06414=1029.447,-36.395,411.260,167.691,43.618,158.080
C06415=1029.454,-36.115,411.246,167.694,43.617,158.080
C06416=1029.461,-35.834,411.232,167.697,43.615,158.080
C06417=1029.467,-35.585,411.218,167.699,43.613,158.080
C06418=1029.473,-35.335,411.206,167.702,43.612,158.080
C06419=1029.479,-35.086,411.192,167.704,43.610,158.080
C06420=1029.485,-34.836,411.180,167.707,43.608,158.080
C06421=1029.491,-34.587,411.167,167.710,43.607,158.079
C06422=1029.498,-34.337,411.153,167.713,43.605,158.079
C06423=1029.504,-34.087,411.140,167.715,43.603,158.079
C06424=1029.510,-33.838,411.127,167.718,43.602,158.079
C06425=1029.516,-33.588,411.115,167.721,43.600,158.079
C06426=1029.522,-33.338,411.101,167.724,43.599,158.079
C06427=1029.528,-33.088,411.089,167.726,43.597,158.079
C06428=1029.534,-32.839,411.075,167.729,43.595,158.079
C06429=1029.541,-32.590,411.062,167.732,43.594,158.079
C06430=1029.547,-32.340,411.050,167.734,43.592,158.079
C06431=1029.553,-32.090,411.036,167.737,43.590,158.079
C06432=1029.560,-31.841,411.023,167.740,43.589,158.079
C06433=1029.565,-31.591,411.010,167.742,43.587,158.079
C06434=1029.572,-31.342,410.997,167.745,43.585,158.078
C06435=1029.578,-31.092,410.984,167.748,43.583,158.078
C06436=1029.584,-30.843,410.971,167.750,43.582,158.078
C06437=1029.591,-30.593,410.957,167.753,43.580,158.078
C06438=1029.597,-30.343,410.944,167.756,43.578,158.078
C06439=1029.603,-30.093,410.932,167.759,43.577,158.078
C06440=1029.609,-29.844,410.918,167.761,43.575,158.078
C06441=1029.615,-29.595,410.905,167.764,43.573,158.078
C06442=1029.621,-29.345,410.893,167.767,43.571,158.078
C06443=1029.628,-29.095,410.879,167.769,43.570,158.078
C06444=1029.634,-28.846,410.866,167.772,43.568,158.078
C06445=1029.640,-28.597,410.852,167.775,43.566,158.078
C06446=1029.646,-28.347,410.840,167.776,43.565,158.077
C06447=1029.653,-28.097,410.826,167.779,43.563,158.077
C06448=1029.659,-27.847,410.813,167.782,43.561,158.077
C06449=1029.666,-27.598,410.800,167.784,43.559,158.077
C06450=1029.671,-27.348,410.787,167.787,43.558,158.077
C06451=1029.678,-27.099,410.774,167.790,43.556,158.077
C06452=1029.684,-26.849,410.760,167.792,43.554,158.077
C06453=1029.690,-26.599,410.746,167.795,43.553,158.077
C06454=1029.696,-26.350,410.733,167.798,43.551,158.077
C06455=1029.702,-26.101,410.720,167.801,43.550,158.077
C06456=1029.709,-25.851,410.706,167.803,43.548,158.077
C06457=1029.714,-25.601,410.693,167.806,43.547,158.077
C06458=1029.721,-25.352,410.680,167.809,43.545,158.077
C06459=1029.727,-25.102,410.666,167.811,43.544,158.076
C06460=1029.734,-24.852,410.653,167.813,43.542,158.076
C06461=1029.739,-24.603,410.639,167.816,43.540,158.076
C06462=1029.745,-24.353,410.626,167.819,43.539,158.076
C06463=1029.751,-24.104,410.612,167.822,43.537,158.076
C06464=1029.758,-23.854,410.599,167.824,43.536,158.076
C06465=1029.764,-23.605,410.585,167.827,43.534,158.076
C06466=1029.770,-23.355,410.572,167.830,43.532,158.076
C06467=1029.776,-23.106,410.558,167.832,43.531,158.076
C06468=1029.782,-22.856,410.544,167.834,43.530,158.076
C06469=1029.788,-22.607,410.531,167.837,43.528,158.076
C06470=1029.795,-22.357,410.518,167.840,43.526,158.076
C06471=1029.802,-22.107,410.504,167.842,43.525,158.076
C06472=1029.807,-21.858,410.490,167.845,43.523,158.076
C06473=1029.813,-21.609,410.477,167.848,43.522,158.075
C06474=1029.820,-21.359,410.463,167.850,43.520,158.075
C06475=1029.826,-21.109,410.449,167.853,43.518,158.075
C06476=1029.832,-20.860,410.436,167.856,43.517,158.075
C06477=1029.839,-20.579,410.420,167.858,43.515,158.075
C06478=1029.846,-20.297,410.406,167.861,43.513,158.075
C06479=1029.853,-20.016,410.390,167.864,43.512,158.075
C06480=1029.860,-19.734,410.374,167.868,43.510,158.075
C06481=1029.867,-19.485,410.361,167.870,43.508,158.075
C06482=1029.873,-19.236,410.348,167.872,43.507,158.075
C06483=1029.879,-18.985,410.333,167.875,43.505,158.075
C06484=1029.885,-18.736,410.320,167.877,43.503,158.075
C06485=1029.891,-18.487,410.307,167.880,43.502,158.075
C06486=1029.897,-18.237,410.293,167.883,43.500,158.074
C06487=1029.904,-17.988,410.279,167.885,43.498,158.074
C06488=1029.911,-17.738,410.265,167.888,43.497,158.074
C06489=1029.916,-17.488,410.251,167.891,43.495,158.074
C06490=1029.922,-17.239,410.238,167.894,43.493,158.074
C06491=1029.929,-16.989,410.224,167.895,43.492,158.074
C06492=1029.935,-16.740,410.210,167.898,43.490,158.074
C06493=1029.942,-16.490,410.196,167.901,43.488,158.074
C06494=1029.948,-16.241,410.183,167.903,43.487,158.074
C06495=1029.955,-15.991,410.169,167.906,43.485,158.074
C06496=1029.960,-15.742,410.155,167.909,43.483,158.074
C06497=1029.967,-15.492,410.142,167.912,43.482,158.074
C06498=1029.973,-15.243,410.127,167.914,43.480,158.073
C06499=1029.979,-14.993,410.114,167.916,43.479,158.073
C06500=1029.985,-14.743,410.099,167.919,43.477,158.073
C06501=1029.992,-14.494,410.085,167.922,43.476,158.073
C06502=1029.998,-14.244,410.071,167.924,43.474,158.073
C06503=1030.003,-13.995,410.057,167.927,43.473,158.073
C06504=1030.010,-13.745,410.043,167.929,43.471,158.073
C06505=1030.016,-13.496,410.029,167.932,43.470,158.073
C06506=1030.023,-13.246,410.016,167.934,43.468,158.073
C06507=1030.029,-12.997,410.001,167.937,43.467,158.073
C06508=1030.035,-12.747,409.988,167.940,43.465,158.073
C06509=1030.041,-12.497,409.973,167.942,43.464,158.073
C06510=1030.047,-12.248,409.959,167.944,43.462,158.073
C06511=1030.053,-11.998,409.945,167.947,43.461,158.073
C06512=1030.059,-11.749,409.931,167.950,43.459,158.072
C06513=1030.066,-11.499,409.917,167.952,43.457,158.072
C06514=1030.072,-11.250,409.902,167.955,43.456,158.072
C06515=1030.079,-11.000,409.889,167.958,43.454,158.072
C06516=1030.084,-10.751,409.875,167.960,43.453,158.072
C06517=1030.091,-10.501,409.860,167.962,43.451,158.072
C06518=1030.097,-10.252,409.847,167.965,43.450,158.072
C06519=1030.103,-10.002,409.832,167.968,43.448,158.072
C06520=1030.109,-9.753,409.818,167.970,43.447,158.072
C06521=1030.116,-9.503,409.804,167.972,43.446,158.072
C06522=1030.121,-9.254,409.790,167.975,43.444,158.072
C06523=1030.128,-9.004,409.775,167.978,43.442,158.072
C06524=1030.134,-8.754,409.761,167.980,43.441,158.072
C06525=1030.141,-8.505,409.747,167.983,43.439,158.072
C06526=1030.147,-8.255,409.733,167.985,43.438,158.071
C06527=1030.153,-8.006,409.718,167.988,43.437,158.071
C06528=1030.160,-7.756,409.705,167.990,43.435,158.071
C06529=1030.165,-7.507,409.690,167.993,43.433,158.071
C06530=1030.172,-7.257,409.676,167.996,43.432,158.071
C06531=1030.178,-7.008,409.662,167.998,43.430,158.071
C06532=1030.184,-6.758,409.648,168.000,43.429,158.071
C06533=1030.191,-6.509,409.633,168.003,43.427,158.071
C06534=1030.197,-6.260,409.619,168.005,43.425,158.071
C06535=1030.204,-6.010,409.605,168.008,43.424,158.071
C06536=1030.210,-5.761,409.590,168.011,43.422,158.071
C06537=1030.216,-5.511,409.576,168.013,43.421,158.071
C06538=1030.223,-5.261,409.562,168.015,43.419,158.070
C06539=1030.229,-5.012,409.547,168.018,43.417,158.070
C06540=1030.235,-4.762,409.534,168.021,43.416,158.070
C06541=1030.242,-4.479,409.517,168.023,43.414,158.070
C06542=1030.249,-4.197,409.501,168.026,43.412,158.070
C06543=1030.257,-3.914,409.485,168.029,43.410,158.070
C06544=1030.264,-3.630,409.469,168.033,43.409,158.070
C06545=1030.270,-3.381,409.454,168.034,43.407,158.070
C06546=1030.276,-3.132,409.439,168.037,43.406,158.070
C06547=1030.282,-2.883,409.424,168.040,43.405,158.070
C06548=1030.288,-2.633,409.409,168.043,43.403,158.070
C06549=1030.294,-2.383,409.395,168.044,43.402,158.070
C06550=1030.300,-2.134,409.381,168.047,43.400,158.070
C06551=1030.307,-1.884,409.366,168.050,43.399,158.070
C06552=1030.312,-1.635,409.351,168.051,43.397,158.069
C06553=1030.319,-1.385,409.336,168.054,43.396,158.069
C06554=1030.325,-1.135,409.322,168.057,43.395,158.069
C06555=1030.331,-0.886,409.307,168.060,43.393,158.069
C06556=1030.337,-0.637,409.292,168.062,43.392,158.069
C06557=1030.343,-0.387,409.277,168.064,43.390,158.069
C06558=1030.349,-0.138,409.263,168.067,43.389,158.069
C06559=1030.356,0.112,409.248,168.070,43.387,158.069
C06560=1030.362,0.361,409.233,168.072,43.386,158.069
C06561=1030.367,0.611,409.219,168.074,43.385,158.069
C06562=1030.374,0.861,409.204,168.077,43.383,158.069
C06563=1030.380,1.110,409.189,168.079,43.382,158.069
C06564=1030.386,1.359,409.175,168.082,43.380,158.069
C06565=1030.393,1.609,409.160,168.084,43.379,158.069
C06566=1030.400,1.858,409.145,168.087,43.377,158.068
C06567=1030.405,2.107,409.131,168.089,43.376,158.068
C06568=1030.412,2.357,409.116,168.091,43.374,158.068
C06569=1030.418,2.607,409.101,168.094,43.373,158.068
C06570=1030.424,2.856,409.086,168.097,43.372,158.068
C06571=1030.430,3.105,409.071,168.099,43.370,158.068
C06572=1030.437,3.355,409.056,168.102,43.369,158.068
C06573=1030.443,3.604,409.042,168.104,43.367,158.068
C06574=1030.449,3.854,409.027,168.106,43.366,158.068
C06575=1030.455,4.103,409.012,168.109,43.364,158.068
C06576=1030.462,4.353,408.997,168.112,43.363,158.068
C06577=1030.468,4.602,408.982,168.114,43.361,158.068
C06578=1030.474,4.852,408.967,168.116,43.360,158.068
C06579=1030.480,5.101,408.953,168.119,43.358,158.068
C06580=1030.486,5.351,408.938,168.122,43.357,158.068
C06581=1030.493,5.600,408.923,168.124,43.355,158.067
C06582=1030.499,5.850,408.908,168.126,43.354,158.067
C06583=1030.505,6.099,408.893,168.129,43.352,158.067
C06584=1030.511,6.349,408.878,168.131,43.351,158.067
C06585=1030.518,6.598,408.863,168.133,43.350,158.067
C06586=1030.524,6.848,408.848,168.136,43.348,158.067
C06587=1030.531,7.098,408.833,168.139,43.347,158.067
C06588=1030.536,7.346,408.819,168.141,43.345,158.067
C06589=1030.543,7.596,408.804,168.143,43.344,158.067
C06590=1030.549,7.846,408.789,168.146,43.342,158.067
C06591=1030.555,8.095,408.774,168.149,43.341,158.067
C06592=1030.562,8.345,408.759,168.151,43.339,158.067
C06593=1030.569,8.594,408.743,168.153,43.338,158.067
C06594=1030.574,8.843,408.729,168.156,43.337,158.067
C06595=1030.581,9.093,408.714,168.158,43.335,158.066
C06596=1030.587,9.342,408.699,168.160,43.333,158.066
C06597=1030.594,9.592,408.684,168.163,43.332,158.066
C06598=1030.600,9.842,408.669,168.166,43.330,158.066
C06599=1030.606,10.091,408.654,168.168,43.329,158.066
C06600=1030.613,10.340,408.638,168.170,43.327,158.066
C06601=1030.619,10.589,408.624,168.173,43.326,158.066
C06602=1030.625,10.839,408.609,168.176,43.324,158.066
C06603=1030.632,11.089,408.594,168.178,43.323,158.066
C06604=1030.638,11.338,408.579,168.180,43.321,158.066
C06605=1030.645,11.624,408.561,168.183,43.319,158.065
C06606=1030.652,11.908,408.544,168.185,43.317,158.065
C06607=1030.659,12.193,408.527,168.189,43.316,158.065
C06608=1030.667,12.478,408.510,168.192,43.314,158.065
C06609=1030.673,12.727,408.494,168.193,43.313,158.065
C06610=1030.680,12.977,408.479,168.196,43.311,158.065
C06611=1030.686,13.227,408.464,168.199,43.310,158.065
C06612=1030.692,13.476,408.449,168.202,43.308,158.065
C06613=1030.699,13.725,408.434,168.203,43.307,158.065
C06614=1030.705,13.974,408.419,168.206,43.306,158.065
C06615=1030.711,14.224,408.404,168.209,43.304,158.065
C06616=1030.717,14.473,408.388,168.211,43.303,158.065
C06617=1030.724,14.723,408.373,168.213,43.301,158.064
C06618=1030.730,14.973,408.358,168.216,43.300,158.064
C06619=1030.737,15.222,408.342,168.218,43.298,158.064
C06620=1030.742,15.472,408.327,168.221,43.297,158.064
C06621=1030.749,15.721,408.311,168.223,43.296,158.064
C06622=1030.755,15.970,408.296,168.225,43.294,158.064
C06623=1030.761,16.220,408.280,168.228,43.293,158.064
C06624=1030.768,16.469,408.265,168.231,43.291,158.064
C06625=1030.774,16.719,408.250,168.232,43.290,158.064
C06626=1030.781,16.968,408.234,168.235,43.288,158.064
C06627=1030.786,17.218,408.219,168.238,43.287,158.064
C06628=1030.793,17.467,408.203,168.239,43.285,158.064
C06629=1030.799,17.717,408.188,168.242,43.284,158.064
C06630=1030.805,17.966,408.172,168.245,43.282,158.064
C06631=1030.812,18.216,408.157,168.247,43.281,158.063
C06632=1030.818,18.465,408.141,168.250,43.280,158.063
C06633=1030.824,18.714,408.126,168.252,43.278,158.063
C06634=1030.830,18.963,408.110,168.254,43.277,158.063
C06635=1030.837,19.213,408.095,168.257,43.275,158.063
C06636=1030.843,19.462,408.080,168.260,43.274,158.063
C06637=1030.849,19.712,408.064,168.261,43.272,158.063
C06638=1030.856,19.961,408.049,168.264,43.271,158.063
C06639=1030.862,20.212,408.033,168.267,43.269,158.063
C06640=1030.869,20.461,408.017,168.269,43.268,158.063
C06641=1030.874,20.711,408.001,168.271,43.267,158.063
C06642=1030.881,20.960,407.986,168.273,43.265,158.063
C06643=1030.887,21.209,407.970,168.276,43.264,158.063
C06644=1030.893,21.459,407.955,168.278,43.262,158.063
C06645=1030.900,21.708,407.939,168.280,43.261,158.062
C06646=1030.906,21.958,407.923,168.283,43.260,158.062
C06647=1030.912,22.207,407.908,168.286,43.258,158.062
C06648=1030.918,22.456,407.891,168.288,43.257,158.062
C06649=1030.925,22.706,407.877,168.290,43.256,158.062
C06650=1030.931,22.955,407.860,168.293,43.254,158.062
C06651=1030.937,23.204,407.845,168.295,43.253,158.062
C06652=1030.943,23.454,407.829,168.298,43.251,158.062
C06653=1030.950,23.703,407.813,168.299,43.250,158.062
C06654=1030.956,23.952,407.797,168.302,43.249,158.062
C06655=1030.962,24.202,407.782,168.305,43.247,158.062
C06656=1030.969,24.451,407.767,168.307,43.246,158.062
C06657=1030.975,24.700,407.750,168.309,43.245,158.062
C06658=1030.981,24.950,407.735,168.312,43.243,158.061
C06659=1030.987,25.199,407.719,168.314,43.242,158.061
C06660=1030.994,25.448,407.703,168.316,43.240,158.061
C06661=1031.000,25.699,407.687,168.319,43.239,158.061
C06662=1031.007,25.948,407.672,168.321,43.237,158.061
C06663=1031.012,26.198,407.656,168.324,43.236,158.061
C06664=1031.019,26.447,407.640,168.326,43.235,158.061
C06665=1031.025,26.696,407.624,168.328,43.233,158.061
C06666=1031.031,26.946,407.609,168.331,43.232,158.061
C06667=1031.037,27.195,407.592,168.333,43.230,158.061
C06668=1031.044,27.444,407.577,168.336,43.229,158.061
C06669=1031.052,27.730,407.558,168.338,43.227,158.061
C06670=1031.059,28.017,407.540,168.341,43.225,158.061
C06671=1031.065,28.303,407.522,168.344,43.224,158.061
C06672=1031.073,28.589,407.503,168.346,43.222,158.060
C06673=1031.079,28.838,407.487,168.349,43.221,158.060
C06674=1031.085,29.088,407.471,168.351,43.220,158.060
C06675=1031.091,29.337,407.455,168.354,43.218,158.060
C06676=1031.098,29.587,407.439,168.355,43.217,158.060
C06677=1031.104,29.837,407.423,168.358,43.215,158.060
C06678=1031.110,30.086,407.407,168.360,43.214,158.060
C06679=1031.116,30.335,407.391,168.363,43.213,158.060
C06680=1031.122,30.584,407.375,168.365,43.211,158.060
C06681=1031.129,30.833,407.359,168.367,43.210,158.060
C06682=1031.135,31.083,407.343,168.370,43.209,158.060
C06683=1031.141,31.333,407.326,168.372,43.208,158.060
C06684=1031.147,31.582,407.310,168.375,43.206,158.060
C06685=1031.154,31.831,407.294,168.377,43.204,158.059
C06686=1031.160,32.080,407.278,168.379,43.203,158.059
C06687=1031.166,32.330,407.262,168.382,43.202,158.059
C06688=1031.173,32.579,407.246,168.384,43.201,158.059
C06689=1031.179,32.829,407.230,168.386,43.199,158.059
C06690=1031.185,33.078,407.213,168.389,43.198,158.059
C06691=1031.191,33.328,407.197,168.391,43.197,158.059
C06692=1031.198,33.577,407.181,168.394,43.195,158.059
C06693=1031.204,33.826,407.165,168.395,43.194,158.059
C06694=1031.210,34.076,407.148,168.398,43.193,158.059
C06695=1031.217,34.325,407.133,168.401,43.191,158.059
C06696=1031.223,34.574,407.117,168.403,43.190,158.059
C06697=1031.229,34.824,407.100,168.405,43.189,158.059
C06698=1031.235,35.074,407.084,168.407,43.187,158.059
C06699=1031.242,35.323,407.068,168.410,43.186,158.059
C06700=1031.248,35.572,407.052,168.413,43.184,158.058
C06701=1031.254,35.822,407.036,168.414,43.183,158.058
C06702=1031.261,36.072,407.019,168.417,43.181,158.058
C06703=1031.268,36.320,407.003,168.419,43.180,158.058
C06704=1031.273,36.569,406.986,168.421,43.178,158.058
C06705=1031.279,36.819,406.970,168.424,43.177,158.058
C06706=1031.286,37.069,406.953,168.426,43.176,158.058
C06707=1031.293,37.318,406.938,168.429,43.174,158.058
C06708=1031.299,37.567,406.921,168.431,43.173,158.058
C06709=1031.305,37.817,406.905,168.433,43.172,158.058
C06710=1031.311,38.066,406.888,168.435,43.170,158.058
C06711=1031.317,38.315,406.872,168.438,43.169,158.058
C06712=1031.323,38.565,406.855,168.441,43.168,158.058
C06713=1031.329,38.814,406.839,168.442,43.166,158.057
C06714=1031.336,39.063,406.822,168.445,43.165,158.057
C06715=1031.342,39.313,406.806,168.447,43.164,158.057
C06716=1031.348,39.562,406.789,168.450,43.162,158.057
C06717=1031.355,39.812,406.773,168.452,43.161,158.057
C06718=1031.361,40.061,406.756,168.454,43.160,158.057
C06719=1031.367,40.310,406.739,168.456,43.158,158.057
C06720=1031.373,40.560,406.723,168.459,43.157,158.057
C06721=1031.379,40.810,406.707,168.462,43.155,158.057
C06722=1031.386,41.058,406.690,168.463,43.154,158.057
C06723=1031.392,41.308,406.673,168.466,43.153,158.057
C06724=1031.398,41.558,406.657,168.468,43.152,158.057
C06725=1031.404,41.806,406.640,168.471,43.150,158.057
C06726=1031.410,42.056,406.623,168.472,43.149,158.057
C06727=1031.417,42.306,406.607,168.475,43.148,158.056
C06728=1031.423,42.555,406.590,168.478,43.146,158.056
C06729=1031.429,42.804,406.574,168.480,43.145,158.056
C06730=1031.436,43.054,406.557,168.482,43.144,158.056
C06731=1031.442,43.303,406.540,168.484,43.143,158.056
C06732=1031.448,43.552,406.524,168.487,43.141,158.056
C06733=1031.455,43.838,406.504,168.490,43.140,158.056
C06734=1031.461,44.125,406.485,168.492,43.139,158.056
C06735=1031.469,44.411,406.466,168.494,43.137,158.056
C06736=1031.476,44.697,406.446,168.497,43.136,158.056
C06737=1031.482,44.946,406.430,168.500,43.134,158.056
C06738=1031.489,45.196,406.412,168.502,43.133,158.056
C06739=1031.494,45.445,406.396,168.504,43.132,158.056
C06740=1031.500,45.694,406.379,168.506,43.131,158.056
C06741=1031.507,45.944,406.362,168.509,43.129,158.056
C06742=1031.513,46.193,406.345,168.511,43.128,158.056
C06743=1031.518,46.442,406.328,168.514,43.127,158.055
C06744=1031.525,46.692,406.311,168.515,43.126,158.055
C06745=1031.531,46.941,406.294,168.518,43.124,158.055
C06746=1031.537,47.190,406.278,168.520,43.123,158.055
C06747=1031.543,47.440,406.260,168.523,43.122,158.055
C06748=1031.549,47.689,406.243,168.524,43.121,158.055
C06749=1031.556,47.938,406.226,168.527,43.119,158.055
C06750=1031.562,48.188,406.210,168.529,43.118,158.055
C06751=1031.568,48.437,406.192,168.532,43.117,158.055
C06752=1031.574,48.687,406.176,168.534,43.116,158.055
C06753=1031.580,48.936,406.159,168.536,43.114,158.055
C06754=1031.587,49.185,406.141,168.538,43.113,158.055
C06755=1031.592,49.435,406.124,168.541,43.112,158.055
C06756=1031.599,49.683,406.107,168.544,43.110,158.055
C06757=1031.605,49.933,406.091,168.546,43.109,158.055
C06758=1031.611,50.182,406.074,168.548,43.108,158.055
C06759=1031.618,50.432,406.056,168.550,43.107,158.054
C06760=1031.624,50.681,406.040,168.553,43.105,158.054
C06761=1031.630,50.930,406.023,168.555,43.104,158.054
C06762=1031.637,51.179,406.005,168.557,43.103,158.054
C06763=1031.642,51.429,405.988,168.559,43.102,158.054
C06764=1031.649,51.678,405.971,168.562,43.100,158.054
C06765=1031.655,51.927,405.954,168.564,43.099,158.054
C06766=1031.661,52.178,405.937,168.567,43.098,158.054
C06767=1031.667,52.426,405.920,168.568,43.096,158.054
C06768=1031.674,52.676,405.903,168.571,43.095,158.054
C06769=1031.680,52.925,405.886,168.573,43.094,158.054
C06770=1031.686,53.175,405.868,168.575,43.092,158.054
C06771=1031.692,53.424,405.851,168.577,43.091,158.054
C06772=1031.699,53.673,405.834,168.580,43.090,158.054
C06773=1031.704,53.923,405.817,168.583,43.088,158.053
C06774=1031.711,54.172,405.800,168.585,43.087,158.053
C06775=1031.717,54.421,405.783,168.587,43.086,158.053
C06776=1031.724,54.670,405.766,168.589,43.084,158.053
C06777=1031.730,54.920,405.749,168.592,43.083,158.053
C06778=1031.736,55.169,405.731,168.594,43.082,158.053
C06779=1031.743,55.418,405.714,168.596,43.080,158.053
C06780=1031.749,55.668,405.697,168.598,43.079,158.053
C06781=1031.755,55.917,405.680,168.601,43.078,158.053
C06782=1031.762,56.167,405.663,168.603,43.076,158.053
C06783=1031.768,56.415,405.646,168.606,43.075,158.053
C06784=1031.774,56.665,405.628,168.607,43.073,158.053
C06785=1031.780,56.914,405.611,168.610,43.072,158.053
C06786=1031.787,57.164,405.594,168.613,43.071,158.053
C06787=1031.793,57.414,405.577,168.615,43.069,158.052
C06788=1031.799,57.662,405.560,168.617,43.068,158.052
C06789=1031.806,57.912,405.542,168.619,43.067,158.052
C06790=1031.812,58.161,405.525,168.622,43.065,158.052
C06791=1031.818,58.410,405.507,168.624,43.064,158.052
C06792=1031.824,58.660,405.491,168.626,43.063,158.052
C06793=1031.831,58.909,405.474,168.628,43.062,158.052
C06794=1031.837,59.159,405.456,168.631,43.061,158.052
C06795=1031.844,59.407,405.439,168.634,43.059,158.052
C06796=1031.850,59.657,405.421,168.635,43.058,158.052
C06797=1031.857,59.943,405.402,168.638,43.056,158.052
C06798=1031.864,60.229,405.382,168.641,43.054,158.051
C06799=1031.872,60.514,405.362,168.644,43.053,158.051
C06800=1031.879,60.800,405.342,168.646,43.051,158.051
C06801=1031.886,61.050,405.325,168.648,43.050,158.051
C06802=1031.891,61.299,405.307,168.651,43.048,158.051
C06803=1031.898,61.548,405.290,168.653,43.047,158.051
C06804=1031.905,61.798,405.273,168.655,43.045,158.051
C06805=1031.911,62.047,405.255,168.658,43.044,158.051
C06806=1031.917,62.296,405.238,168.660,43.043,158.051
C06807=1031.924,62.546,405.220,168.662,43.041,158.051
C06808=1031.930,62.795,405.203,168.664,43.040,158.051
C06809=1031.937,63.044,405.186,168.667,43.039,158.051
C06810=1031.944,63.293,405.168,168.669,43.038,158.051
C06811=1031.949,63.542,405.151,168.671,43.036,158.050
C06812=1031.956,63.792,405.133,168.673,43.035,158.050
C06813=1031.962,64.042,405.115,168.676,43.034,158.050
C06814=1031.968,64.290,405.098,168.679,43.032,158.050
C06815=1031.974,64.540,405.080,168.681,43.031,158.050
C06816=1031.980,64.789,405.063,168.683,43.030,158.050
C06817=1031.987,65.039,405.046,168.685,43.029,158.050
C06818=1031.993,65.288,405.027,168.688,43.027,158.050
C06819=1032.000,65.536,405.010,168.690,43.026,158.050
C06820=1032.006,65.786,404.992,168.693,43.025,158.050
C06821=1032.012,66.036,404.974,168.694,43.023,158.050
C06822=1032.018,66.285,404.957,168.697,43.022,158.050
C06823=1032.024,66.534,404.939,168.699,43.021,158.050
C06824=1032.031,66.783,404.920,168.701,43.019,158.049
C06825=1032.037,67.032,404.904,168.703,43.018,158.049
C06826=1032.043,67.282,404.886,168.706,43.017,158.049
C06827=1032.049,67.532,404.868,168.708,43.016,158.049
C06828=1032.055,67.780,404.851,168.711,43.014,158.049
C06829=1032.062,68.030,404.832,168.712,43.013,158.049
C06830=1032.068,68.279,404.814,168.715,43.012,158.049
C06831=1032.075,68.529,404.797,168.717,43.010,158.049
C06832=1032.080,68.778,404.779,168.720,43.009,158.049
C06833=1032.086,69.028,404.761,168.722,43.008,158.049
C06834=1032.094,69.276,404.743,168.724,43.007,158.049
C06835=1032.099,69.525,404.726,168.726,43.005,158.049
C06836=1032.105,69.775,404.708,168.729,43.004,158.049
C06837=1032.112,70.024,404.689,168.731,43.003,158.049
C06838=1032.118,70.274,404.671,168.734,43.002,158.049
C06839=1032.124,70.523,404.654,168.735,43.000,158.048
C06840=1032.130,70.772,404.636,168.738,42.999,158.048
C06841=1032.136,71.022,404.618,168.740,42.998,158.048
C06842=1032.142,71.271,404.600,168.743,42.997,158.048
C06843=1032.148,71.520,404.581,168.744,42.995,158.048
C06844=1032.155,71.769,404.564,168.747,42.994,158.048
C06845=1032.161,72.019,404.546,168.749,42.993,158.048
C06846=1032.167,72.267,404.528,168.752,42.992,158.048
C06847=1032.173,72.517,404.510,168.754,42.990,158.048
C06848=1032.179,72.767,404.492,168.756,42.989,158.048
C06849=1032.186,73.016,404.473,168.758,42.988,158.048
C06850=1032.192,73.265,404.456,168.761,42.986,158.048
C06851=1032.199,73.514,404.438,168.763,42.985,158.048
C06852=1032.205,73.764,404.420,168.766,42.984,158.048
C06853=1032.211,74.013,404.401,168.767,42.983,158.048
C06854=1032.217,74.262,404.384,168.770,42.981,158.047
C06855=1032.223,74.511,404.366,168.772,42.980,158.047
C06856=1032.230,74.760,404.348,168.775,42.979,158.047
C06857=1032.236,75.010,404.330,168.776,42.978,158.047
C06858=1032.242,75.259,404.311,168.779,42.977,158.047
C06859=1032.248,75.508,404.293,168.781,42.976,158.047
C06860=1032.254,75.757,404.275,168.784,42.974,158.047
C06861=1032.262,76.043,404.254,168.786,42.973,158.047
C06862=1032.269,76.329,404.234,168.789,42.971,158.047
C06863=1032.276,76.615,404.212,168.791,42.970,158.047
C06864=1032.283,76.900,404.192,168.794,42.969,158.047
C06865=1032.289,77.149,404.173,168.797,42.967,158.047
C06866=1032.296,77.399,404.155,168.798,42.966,158.047
C06867=1032.301,77.647,404.137,168.801,42.965,158.047
C06868=1032.308,77.897,404.119,168.803,42.964,158.047
C06869=1032.314,78.146,404.100,168.806,42.962,158.047
C06870=1032.320,78.395,404.082,168.807,42.961,158.046
C06871=1032.327,78.645,404.064,168.810,42.960,158.046
C06872=1032.333,78.894,404.045,168.812,42.959,158.046
C06873=1032.338,79.143,404.028,168.815,42.958,158.046
C06874=1032.345,79.392,404.009,168.817,42.957,158.046
C06875=1032.351,79.642,403.990,168.820,42.955,158.046
C06876=1032.357,79.892,403.972,168.821,42.954,158.046
C06877=1032.363,80.141,403.953,168.824,42.953,158.046
C06878=1032.370,80.390,403.934,168.826,42.952,158.046
C06879=1032.375,80.639,403.917,168.829,42.950,158.046
C06880=1032.382,80.888,403.898,168.831,42.949,158.046
C06881=1032.388,81.137,403.880,168.833,42.948,158.046
C06882=1032.394,81.386,403.861,168.835,42.947,158.046
C06883=1032.400,81.636,403.842,168.838,42.945,158.046
C06884=1032.406,81.885,403.824,168.840,42.944,158.046
C06885=1032.412,82.134,403.805,168.843,42.943,158.046
C06886=1032.418,82.384,403.788,168.844,42.942,158.046
C06887=1032.425,82.633,403.769,168.847,42.941,158.045
C06888=1032.431,82.882,403.750,168.849,42.940,158.045
C06889=1032.437,83.131,403.732,168.852,42.938,158.045
C06890=1032.443,83.380,403.712,168.854,42.937,158.045
C06891=1032.449,83.630,403.694,168.856,42.936,158.045
C06892=1032.456,83.879,403.676,168.858,42.935,158.045
C06893=1032.462,84.128,403.657,168.861,42.933,158.045
C06894=1032.468,84.377,403.638,168.863,42.932,158.045
C06895=1032.474,84.627,403.621,168.865,42.931,158.045
C06896=1032.480,84.876,403.602,168.867,42.930,158.045
C06897=1032.486,85.125,403.583,168.870,42.929,158.045
C06898=1032.493,85.374,403.564,168.872,42.928,158.045
C06899=1032.499,85.623,403.546,168.875,42.926,158.045
C06900=1032.505,85.872,403.527,168.876,42.925,158.045
C06901=1032.512,86.122,403.509,168.879,42.924,158.045
C06902=1032.518,86.371,403.490,168.881,42.923,158.045
C06903=1032.524,86.620,403.472,168.884,42.921,158.045
C06904=1032.530,86.870,403.453,168.885,42.920,158.044
C06905=1032.536,87.119,403.434,168.888,42.919,158.044
C06906=1032.543,87.368,403.415,168.890,42.918,158.044
C06907=1032.549,87.617,403.397,168.893,42.916,158.044
C06908=1032.555,87.867,403.379,168.895,42.915,158.044
C06909=1032.562,88.116,403.360,168.897,42.914,158.044
C06910=1032.568,88.366,403.341,168.899,42.913,158.044
C06911=1032.574,88.615,403.322,168.902,42.912,158.044
C06912=1032.580,88.864,403.304,168.904,42.910,158.044
C06913=1032.587,89.113,403.285,168.907,42.909,158.044
C06914=1032.593,89.362,403.266,168.908,42.908,158.044
C06915=1032.600,89.611,403.248,168.911,42.907,158.044
C06916=1032.605,89.861,403.228,168.913,42.905,158.044
C06917=1032.612,90.110,403.210,168.916,42.904,158.044
C06918=1032.618,90.359,403.191,168.918,42.903,158.043
C06919=1032.624,90.608,403.172,168.920,42.902,158.043
C06920=1032.630,90.857,403.153,168.922,42.901,158.043
C06921=1032.636,91.107,403.134,168.925,42.900,158.043
C06922=1032.642,91.356,403.115,168.927,42.899,158.043
C06923=1032.648,91.605,403.096,168.930,42.897,158.043
C06924=1032.655,91.854,403.077,168.931,42.896,158.043
C06925=1032.661,92.139,403.055,168.934,42.895,158.043
C06926=1032.668,92.425,403.034,168.937,42.893,158.043
C06927=1032.675,92.711,403.012,168.940,42.892,158.043
C06928=1032.682,92.996,402.991,168.943,42.891,158.043
C06929=1032.689,93.245,402.971,168.944,42.890,158.043
C06930=1032.694,93.494,402.952,168.947,42.888,158.043
C06931=1032.701,93.743,402.933,168.949,42.887,158.043
C06932=1032.706,93.993,402.914,168.952,42.886,158.043
C06933=1032.713,94.242,402.895,168.954,42.885,158.043
C06934=1032.719,94.491,402.876,168.956,42.883,158.043
C06935=1032.726,94.741,402.857,168.958,42.882,158.043
C06936=1032.732,94.990,402.838,168.961,42.881,158.043
C06937=1032.738,95.239,402.819,168.963,42.880,158.042
C06938=1032.744,95.488,402.800,168.966,42.879,158.042
C06939=1032.750,95.738,402.781,168.967,42.878,158.042
C06940=1032.757,95.987,402.762,168.970,42.876,158.042
C06941=1032.763,96.236,402.742,168.972,42.875,158.042
C06942=1032.769,96.485,402.723,168.975,42.874,158.042
C06943=1032.775,96.734,402.704,168.977,42.873,158.042
C06944=1032.781,96.983,402.685,168.979,42.871,158.042
C06945=1032.787,97.233,402.666,168.981,42.870,158.042
C06946=1032.794,97.481,402.647,168.984,42.869,158.042
C06947=1032.799,97.731,402.628,168.987,42.868,158.042
C06948=1032.806,97.981,402.609,168.989,42.867,158.042
C06949=1032.812,98.230,402.589,168.992,42.866,158.042
C06950=1032.819,98.478,402.570,168.993,42.864,158.042
C06951=1032.824,98.728,402.551,168.996,42.863,158.042
C06952=1032.831,98.977,402.532,168.998,42.862,158.042
C06953=1032.837,99.226,402.512,169.001,42.861,158.042
C06954=1032.843,99.475,402.493,169.002,42.860,158.042
C06955=1032.850,99.724,402.475,169.005,42.858,158.041
C06956=1032.856,99.974,402.455,169.007,42.857,158.041
C06957=1032.862,100.223,402.435,169.010,42.856,158.041
C06958=1032.868,100.472,402.417,169.012,42.855,158.041
C06959=1032.874,100.721,402.397,169.014,42.854,158.041
C06960=1032.880,100.970,402.377,169.016,42.853,158.041
C06961=1032.886,101.220,402.358,169.019,42.852,158.041
C06962=1032.892,101.468,402.339,169.021,42.851,158.041
C06963=1032.899,101.718,402.319,169.024,42.850,158.041
C06964=1032.905,101.967,402.299,169.026,42.849,158.041
C06965=1032.910,102.217,402.280,169.029,42.848,158.041
C06966=1032.917,102.465,402.261,169.030,42.846,158.041
C06967=1032.923,102.715,402.241,169.033,42.845,158.041
C06968=1032.929,102.963,402.221,169.035,42.844,158.041
C06969=1032.934,103.213,402.202,169.038,42.843,158.041
C06970=1032.942,103.462,402.182,169.039,42.842,158.041
C06971=1032.948,103.712,402.163,169.042,42.841,158.041
C06972=1032.954,103.960,402.143,169.044,42.840,158.041
C06973=1032.959,104.210,402.124,169.047,42.839,158.041
C06974=1032.966,104.458,402.105,169.049,42.838,158.041
C06975=1032.972,104.708,402.085,169.052,42.836,158.041
C06976=1032.978,104.957,402.065,169.055,42.835,158.041
C06977=1032.984,105.207,402.046,169.056,42.834,158.040
C06978=1032.990,105.455,402.026,169.059,42.832,158.040
C06979=1032.996,105.705,402.007,169.061,42.831,158.040
C06980=1033.002,105.953,401.987,169.064,42.830,158.040
C06981=1033.009,106.204,401.968,169.065,42.829,158.040
C06982=1033.015,106.452,401.948,169.068,42.828,158.040
C06983=1033.021,106.701,401.928,169.070,42.827,158.040
C06984=1033.027,106.950,401.909,169.073,42.826,158.040
C06985=1033.036,107.279,401.883,169.076,42.824,158.040
C06986=1033.044,107.608,401.857,169.079,42.823,158.040
C06987=1033.051,107.936,401.831,169.082,42.821,158.040
C06988=1033.060,108.266,401.805,169.085,42.820,158.040
C06989=1033.070,108.678,401.773,169.089,42.818,158.040
C06990=1033.080,109.089,401.741,169.093,42.816,158.040
C06991=1033.086,109.338,401.721,169.095,42.815,158.040
C06992=1033.093,109.587,401.700,169.098,42.814,158.040
C06993=1033.099,109.837,401.681,169.100,42.813,158.040
C06994=1033.105,110.086,401.661,169.103,42.812,158.040
C06995=1033.111,110.334,401.642,169.104,42.810,158.039
C06996=1033.118,110.584,401.622,169.107,42.809,158.039
C06997=1033.124,110.833,401.602,169.110,42.808,158.039
C06998=1033.130,111.082,401.582,169.112,42.807,158.039
C06999=1033.136,111.331,401.562,169.115,42.806,158.039
C07000=1033.142,111.581,401.543,169.117,42.805,158.039
C07001=1033.148,111.830,401.523,169.119,42.804,158.039
C07002=1033.154,112.078,401.503,169.121,42.803,158.039
C07003=1033.161,112.328,401.482,169.124,42.801,158.039
C07004=1033.167,112.577,401.462,169.126,42.800,158.039
C07005=1033.172,112.826,401.443,169.129,42.799,158.039
C07006=1033.179,113.076,401.423,169.131,42.798,158.039
C07007=1033.185,113.324,401.403,169.133,42.797,158.039
C07008=1033.191,113.573,401.383,169.135,42.796,158.039
C07009=1033.197,113.823,401.362,169.138,42.795,158.039
C07010=1033.203,114.072,401.342,169.140,42.794,158.039
C07011=1033.209,114.321,401.322,169.143,42.793,158.039
C07012=1033.215,114.570,401.302,169.146,42.792,158.039
C07013=1033.221,114.819,401.282,169.147,42.791,158.039
C07014=1033.226,115.069,401.262,169.150,42.790,158.039
C07015=1033.232,115.318,401.242,169.152,42.789,158.039
C07016=1033.239,115.567,401.222,169.155,42.788,158.039
C07017=1033.245,115.816,401.202,169.157,42.787,158.039
C07018=1033.250,116.065,401.181,169.160,42.786,158.039
C07019=1033.256,116.314,401.161,169.162,42.785,158.039
C07020=1033.263,116.563,401.141,169.164,42.784,158.039
C07021=1033.269,116.812,401.121,169.166,42.783,158.039
C07022=1033.275,117.061,401.101,169.169,42.782,158.039
C07023=1033.281,117.311,401.080,169.171,42.781,158.039
C07024=1033.286,117.560,401.060,169.174,42.780,158.038
C07025=1033.292,117.808,401.040,169.176,42.779,158.038
C07026=1033.299,118.057,401.019,169.178,42.778,158.038
C07027=1033.305,118.306,400.999,169.180,42.777,158.038
C07028=1033.311,118.556,400.978,169.183,42.775,158.038
C07029=1033.317,118.805,400.958,169.186,42.774,158.038
C07030=1033.323,119.054,400.938,169.188,42.773,158.038
C07031=1033.329,119.303,400.917,169.191,42.772,158.038
C07032=1033.335,119.552,400.897,169.193,42.772,158.038
C07033=1033.341,119.801,400.878,169.196,42.771,158.038
C07034=1033.348,120.051,400.857,169.197,42.770,158.038
C07035=1033.353,120.300,400.837,169.200,42.769,158.038
C07036=1033.360,120.549,400.816,169.202,42.768,158.038
C07037=1033.366,120.798,400.796,169.205,42.767,158.038
C07038=1033.372,121.046,400.776,169.208,42.765,158.038
C07039=1033.378,121.296,400.755,169.210,42.764,158.038
C07040=1033.384,121.545,400.735,169.212,42.763,158.038
C07041=1033.390,121.794,400.714,169.214,42.762,158.038
C07042=1033.396,122.043,400.695,169.217,42.761,158.038
C07043=1033.402,122.292,400.674,169.219,42.760,158.038
C07044=1033.408,122.541,400.653,169.222,42.759,158.038
C07045=1033.414,122.790,400.633,169.225,42.758,158.038
C07046=1033.421,123.040,400.613,169.226,42.757,158.038
C07047=1033.426,123.289,400.592,169.229,42.756,158.038
C07048=1033.433,123.538,400.572,169.231,42.755,158.038
C07049=1033.439,123.786,400.551,169.234,42.754,158.038
C07050=1033.446,124.036,400.531,169.237,42.753,158.038
C07051=1033.453,124.321,400.507,169.240,42.751,158.038
C07052=1033.459,124.606,400.484,169.242,42.750,158.038
C07053=1033.466,124.892,400.461,169.245,42.749,158.038
C07054=1033.473,125.177,400.437,169.248,42.747,158.038
C07055=1033.480,125.426,400.416,169.250,42.747,158.038
C07056=1033.486,125.675,400.396,169.253,42.746,158.038
C07057=1033.492,125.925,400.375,169.255,42.745,158.038
C07058=1033.498,126.174,400.355,169.258,42.744,158.038
C07059=1033.505,126.423,400.334,169.260,42.743,158.038
C07060=1033.511,126.671,400.314,169.262,42.742,158.037
C07061=1033.516,126.921,400.293,169.265,42.741,158.037
C07062=1033.523,127.169,400.273,169.267,42.740,158.037
C07063=1033.529,127.419,400.252,169.270,42.738,158.037
C07064=1033.535,127.669,400.231,169.273,42.737,158.037
C07065=1033.541,127.917,400.211,169.274,42.736,158.037
C07066=1033.548,128.167,400.190,169.277,42.735,158.037
C07067=1033.554,128.415,400.171,169.280,42.733,158.037
C07068=1033.560,128.665,400.149,169.282,42.732,158.037
C07069=1033.566,128.913,400.129,169.285,42.731,158.037
C07070=1033.573,129.163,400.109,169.287,42.730,158.037
C07071=1033.578,129.411,400.087,169.289,42.729,158.037
C07072=1033.585,129.661,400.067,169.292,42.728,158.037
C07073=1033.592,129.910,400.046,169.295,42.727,158.037
C07074=1033.597,130.159,400.025,169.297,42.726,158.037
C07075=1033.604,130.408,400.005,169.300,42.725,158.037
C07076=1033.610,130.657,399.984,169.301,42.724,158.037
C07077=1033.616,130.906,399.964,169.304,42.723,158.037
C07078=1033.623,131.155,399.942,169.307,42.722,158.037
C07079=1033.628,131.404,399.922,169.309,42.721,158.037
C07080=1033.634,131.654,399.900,169.312,42.720,158.037
C07081=1033.640,131.902,399.880,169.315,42.719,158.037
C07082=1033.646,132.152,399.859,169.317,42.718,158.037
C07083=1033.653,132.400,399.838,169.320,42.717,158.037
C07084=1033.658,132.650,399.817,169.322,42.716,158.037
C07085=1033.664,132.898,399.796,169.324,42.715,158.037
C07086=1033.671,133.148,399.775,169.327,42.714,158.037
C07087=1033.677,133.397,399.754,169.329,42.713,158.037
C07088=1033.683,133.645,399.733,169.332,42.712,158.037
C07089=1033.689,133.895,399.712,169.334,42.711,158.037
C07090=1033.694,134.143,399.691,169.337,42.710,158.037
C07091=1033.701,134.393,399.671,169.340,42.710,158.037
C07092=1033.707,134.642,399.649,169.341,42.709,158.037
C07093=1033.713,134.891,399.628,169.344,42.707,158.037
C07094=1033.719,135.140,399.607,169.347,42.706,158.037
C07095=1033.726,135.389,399.586,169.349,42.705,158.037
C07096=1033.732,135.638,399.565,169.352,42.704,158.037
C07097=1033.738,135.887,399.544,169.355,42.703,158.037
C07098=1033.743,136.136,399.523,169.357,42.703,158.037
C07099=1033.750,136.385,399.502,169.360,42.702,158.037
C07100=1033.756,136.635,399.481,169.362,42.700,158.037
C07101=1033.762,136.883,399.460,169.364,42.699,158.037
C07102=1033.769,137.132,399.439,169.367,42.698,158.037
C07103=1033.775,137.381,399.417,169.370,42.697,158.036
C07104=1033.780,137.630,399.396,169.372,42.697,158.037
C07105=1033.787,137.879,399.375,169.375,42.696,158.037
C07106=1033.793,138.128,399.354,169.377,42.695,158.036
C07107=1033.799,138.377,399.333,169.379,42.694,158.036
C07108=1033.805,138.626,399.311,169.382,42.693,158.036
C07109=1033.811,138.876,399.291,169.384,42.692,158.036
C07110=1033.817,139.124,399.269,169.387,42.691,158.037
C07111=1033.823,139.373,399.248,169.390,42.690,158.037
C07112=1033.829,139.623,399.226,169.392,42.689,158.036
C07113=1033.835,139.871,399.205,169.395,42.688,158.036
C07114=1033.841,140.120,399.183,169.398,42.687,158.037
C07115=1033.848,140.406,399.159,169.401,42.686,158.037
C07116=1033.855,140.691,399.135,169.403,42.685,158.037
C07117=1033.862,140.976,399.110,169.406,42.684,158.036
C07118=1033.869,141.262,399.086,169.409,42.683,158.036
C07119=1033.874,141.510,399.064,169.412,42.682,158.037
C07120=1033.881,141.759,399.043,169.414,42.681,158.037
C07121=1033.887,142.009,399.022,169.417,42.680,158.037
C07122=1033.893,142.257,399.000,169.420,42.679,158.036
C07123=1033.899,142.506,398.979,169.422,42.679,158.037
C07124=1033.905,142.755,398.957,169.425,42.678,158.037
C07125=1033.911,143.005,398.935,169.427,42.677,158.037
C07126=1033.917,143.253,398.914,169.429,42.676,158.036
C07127=1033.923,143.502,398.892,169.432,42.674,158.036
C07128=1033.930,143.751,398.871,169.435,42.674,158.037
C07129=1033.936,144.000,398.850,169.437,42.673,158.037
C07130=1033.942,144.249,398.829,169.440,42.672,158.036
C07131=1033.948,144.498,398.807,169.443,42.671,158.036
C07132=1033.954,144.747,398.785,169.445,42.670,158.037
C07133=1033.960,144.997,398.764,169.447,42.669,158.037
C07134=1033.966,145.246,398.742,169.450,42.668,158.037
C07135=1033.972,145.494,398.721,169.453,42.667,158.036
C07136=1033.978,145.744,398.699,169.455,42.667,158.037
C07137=1033.984,145.993,398.677,169.458,42.666,158.037
C07138=1033.991,146.242,398.656,169.461,42.664,158.037
C07139=1033.997,146.491,398.635,169.463,42.663,158.036
C07140=1034.003,146.739,398.613,169.466,42.663,158.037
C07141=1034.009,146.988,398.591,169.469,42.662,158.037
C07142=1034.015,147.237,398.569,169.470,42.661,158.037
C07143=1034.021,147.487,398.547,169.473,42.660,158.037
C07144=1034.027,147.736,398.526,169.476,42.659,158.037
C07145=1034.033,147.984,398.504,169.479,42.658,158.037
C07146=1034.039,148.233,398.482,169.481,42.658,158.037
C07147=1034.045,148.482,398.460,169.484,42.657,158.037
C07148=1034.051,148.731,398.439,169.487,42.656,158.037
C07149=1034.058,148.981,398.417,169.489,42.655,158.037
C07150=1034.063,149.229,398.396,169.492,42.654,158.037
C07151=1034.070,149.478,398.374,169.495,42.653,158.037
C07152=1034.076,149.727,398.352,169.498,42.652,158.037
C07153=1034.081,149.976,398.330,169.499,42.652,158.037
C07154=1034.088,150.225,398.307,169.502,42.651,158.037
C07155=1034.094,150.474,398.286,169.505,42.650,158.037
C07156=1034.100,150.723,398.264,169.507,42.649,158.037
C07157=1034.106,150.972,398.243,169.510,42.648,158.037
C07158=1034.112,151.220,398.220,169.513,42.647,158.037
C07159=1034.118,151.470,398.198,169.516,42.646,158.037
C07160=1034.124,151.719,398.177,169.518,42.646,158.037
C07161=1034.130,151.968,398.154,169.521,42.645,158.037
C07162=1034.136,152.217,398.133,169.524,42.644,158.037
C07163=1034.142,152.466,398.111,169.527,42.643,158.037
C07164=1034.149,152.715,398.089,169.528,42.642,158.037
C07165=1034.154,152.964,398.067,169.531,42.642,158.037
C07166=1034.160,153.212,398.044,169.534,42.641,158.037
C07167=1034.166,153.461,398.023,169.537,42.639,158.037
C07168=1034.173,153.711,398.001,169.539,42.639,158.037
C07169=1034.179,153.959,397.979,169.542,42.638,158.037
C07170=1034.184,154.209,397.957,169.545,42.637,158.037
C07171=1034.191,154.457,397.934,169.548,42.636,158.037
C07172=1034.197,154.706,397.913,169.550,42.635,158.037
C07173=1034.203,154.955,397.890,169.553,42.635,158.037
C07174=1034.209,155.205,397.868,169.556,42.634,158.037
C07175=1034.215,155.453,397.846,169.559,42.633,158.037
C07176=1034.222,155.702,397.824,169.561,42.632,158.037
C07177=1034.227,155.951,397.801,169.564,42.632,158.037
C07178=1034.233,156.200,397.780,169.566,42.631,158.037
C07179=1034.240,156.485,397.754,169.569,42.630,158.037
C07180=1034.247,156.770,397.729,169.572,42.629,158.037
C07181=1034.254,157.054,397.703,169.575,42.628,158.037
C07182=1034.260,157.340,397.678,169.578,42.628,158.038
C07183=1034.267,157.588,397.656,169.581,42.626,158.038
C07184=1034.273,157.837,397.633,169.584,42.625,158.038
C07185=1034.279,158.086,397.611,169.587,42.625,158.038
C07186=1034.285,158.335,397.589,169.590,42.624,158.038
C07187=1034.291,158.584,397.567,169.592,42.623,158.038
C07188=1034.297,158.833,397.544,169.595,42.622,158.038
C07189=1034.304,159.081,397.522,169.598,42.622,158.038
C07190=1034.309,159.331,397.500,169.600,42.621,158.038
C07191=1034.316,159.580,397.477,169.604,42.620,158.038
C07192=1034.322,159.829,397.456,169.605,42.619,158.038
C07193=1034.327,160.078,397.433,169.608,42.619,158.038
C07194=1034.333,160.327,397.410,169.611,42.618,158.038
C07195=1034.340,160.575,397.387,169.614,42.617,158.038
C07196=1034.345,160.824,397.364,169.616,42.617,158.038
C07197=1034.351,161.074,397.342,169.619,42.616,158.038
C07198=1034.356,161.322,397.319,169.622,42.615,158.038
C07199=1034.363,161.571,397.297,169.625,42.615,158.038
C07200=1034.369,161.820,397.274,169.627,42.614,158.038
C07201=1034.374,162.069,397.251,169.630,42.613,158.038
C07202=1034.380,162.318,397.228,169.633,42.613,158.038
C07203=1034.386,162.567,397.205,169.636,42.612,158.039
C07204=1034.392,162.816,397.184,169.638,42.611,158.039
C07205=1034.398,163.065,397.161,169.641,42.611,158.039
C07206=1034.403,163.314,397.138,169.644,42.610,158.039
C07207=1034.409,163.563,397.115,169.647,42.609,158.039
C07208=1034.416,163.811,397.092,169.649,42.609,158.039
C07209=1034.421,164.060,397.069,169.652,42.608,158.039
C07210=1034.427,164.309,397.046,169.655,42.607,158.039
C07211=1034.433,164.558,397.023,169.658,42.607,158.039
C07212=1034.439,164.806,397.001,169.661,42.606,158.039
C07213=1034.445,165.055,396.978,169.663,42.605,158.039
C07214=1034.451,165.304,396.955,169.666,42.605,158.039
C07215=1034.457,165.553,396.932,169.669,42.604,158.039
C07216=1034.464,165.802,396.910,169.672,42.603,158.039
C07217=1034.469,166.051,396.887,169.675,42.603,158.039
C07218=1034.475,166.300,396.864,169.677,42.602,158.040
C07219=1034.481,166.549,396.841,169.680,42.602,158.040
C07220=1034.487,166.798,396.818,169.683,42.601,158.040
C07221=1034.493,167.047,396.795,169.686,42.600,158.040
C07222=1034.499,167.295,396.773,169.689,42.600,158.040
C07223=1034.504,167.544,396.750,169.692,42.599,158.040
C07224=1034.510,167.793,396.727,169.694,42.598,158.040
C07225=1034.516,168.042,396.704,169.697,42.598,158.040
C07226=1034.523,168.291,396.681,169.699,42.597,158.040
C07227=1034.529,168.540,396.658,169.703,42.596,158.040
C07228=1034.534,168.789,396.635,169.706,42.596,158.040
C07229=1034.540,169.038,396.612,169.709,42.595,158.040
C07230=1034.546,169.287,396.589,169.710,42.594,158.040
C07231=1034.553,169.535,396.566,169.713,42.594,158.040
C07232=1034.558,169.784,396.543,169.717,42.594,158.041
C07233=1034.565,170.033,396.520,169.719,42.592,158.040
C07234=1034.570,170.282,396.497,169.722,42.592,158.041
C07235=1034.576,170.531,396.474,169.725,42.591,158.041
C07236=1034.583,170.780,396.452,169.728,42.590,158.041
C07237=1034.588,171.029,396.429,169.730,42.590,158.041
C07238=1034.595,171.278,396.405,169.733,42.590,158.041
C07239=1034.601,171.527,396.382,169.736,42.589,158.041
C07240=1034.607,171.776,396.359,169.739,42.588,158.041
C07241=1034.613,172.024,396.336,169.742,42.587,158.041
C07242=1034.619,172.273,396.313,169.745,42.587,158.041
C07243=1034.626,172.558,396.286,169.748,42.586,158.041
C07244=1034.633,172.842,396.260,169.751,42.585,158.041
C07245=1034.640,173.126,396.234,169.755,42.585,158.041
C07246=1034.647,173.411,396.207,169.758,42.584,158.042
C07247=1034.653,173.660,396.184,169.761,42.583,158.042
C07248=1034.659,173.908,396.161,169.764,42.583,158.042
C07249=1034.665,174.157,396.138,169.767,42.582,158.042
C07250=1034.671,174.406,396.114,169.770,42.581,158.042
C07251=1034.677,174.655,396.091,169.773,42.581,158.042
C07252=1034.683,174.904,396.068,169.776,42.580,158.042
C07253=1034.690,175.153,396.044,169.779,42.580,158.042
C07254=1034.696,175.402,396.022,169.781,42.579,158.042
C07255=1034.702,175.650,395.998,169.784,42.578,158.042
C07256=1034.708,175.899,395.976,169.787,42.578,158.042
C07257=1034.714,176.148,395.952,169.790,42.577,158.042
C07258=1034.720,176.397,395.929,169.793,42.576,158.042
C07259=1034.726,176.646,395.906,169.796,42.576,158.043
C07260=1034.733,176.895,395.883,169.799,42.575,158.043
C07261=1034.739,177.143,395.859,169.802,42.575,158.043
C07262=1034.745,177.392,395.836,169.805,42.574,158.043
C07263=1034.751,177.641,395.812,169.808,42.573,158.043
C07264=1034.757,177.890,395.789,169.811,42.573,158.043
C07265=1034.764,178.139,395.765,169.814,42.572,158.043
C07266=1034.770,178.388,395.743,169.817,42.571,158.043
C07267=1034.776,178.636,395.720,169.820,42.570,158.043
C07268=1034.783,178.885,395.696,169.823,42.570,158.043
C07269=1034.788,179.134,395.673,169.826,42.570,158.043
C07270=1034.794,179.383,395.649,169.829,42.568,158.043
C07271=1034.801,179.632,395.626,169.832,42.568,158.043
C07272=1034.807,179.880,395.602,169.835,42.567,158.044
C07273=1034.813,180.130,395.579,169.838,42.567,158.044
C07274=1034.820,180.378,395.556,169.841,42.566,158.044
C07275=1034.826,180.627,395.532,169.844,42.565,158.044
C07276=1034.832,180.876,395.509,169.847,42.565,158.044
C07277=1034.838,181.124,395.485,169.850,42.564,158.044
C07278=1034.845,181.374,395.462,169.853,42.564,158.044
C07279=1034.851,181.622,395.438,169.856,42.563,158.044
C07280=1034.857,181.872,395.415,169.859,42.562,158.044
C07281=1034.864,182.120,395.392,169.862,42.562,158.044
C07282=1034.870,182.369,395.368,169.865,42.561,158.044
C07283=1034.876,182.617,395.345,169.868,42.561,158.045
C07284=1034.883,182.866,395.321,169.871,42.560,158.045
C07285=1034.888,183.115,395.298,169.874,42.559,158.045
C07286=1034.895,183.364,395.274,169.877,42.559,158.045
C07287=1034.900,183.613,395.250,169.880,42.558,158.045
